KUKA KRL program: MyProgram_329().src

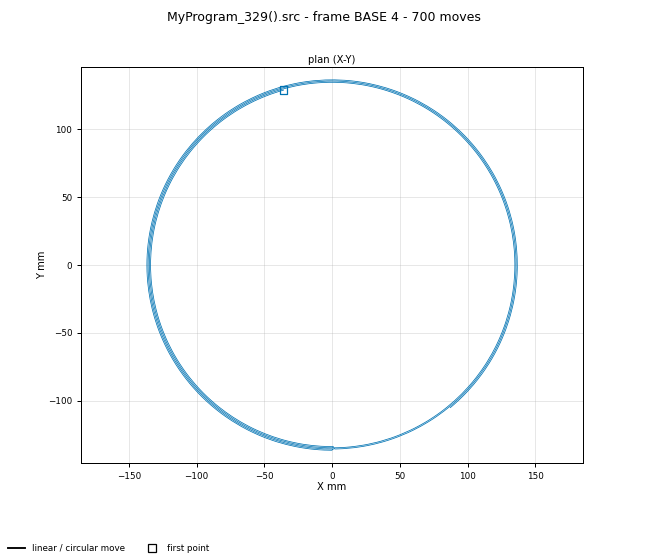
[picture p0: tool path of MyProgram_329().src in frame BASE 4, 700 of 700 moves have a stored position in this frame; points joined in program order, loops and branches not executed]
&ACCESS RVP
&REL 1
&PARAM TEMPLATE = C:\KRC\Roboter\Template\vorgabe
&PARAM EDITMASK = *
DEF MyProgram_329()
; ---- Setting reference (Base) ----
$BASE = BASE_DATA[4]

; --------------------------
; ---- Setting tool (TCP) ----
$TOOL = TOOL_DATA[3]
; --------------------------

$VEL.CP = VEL_APROX_PRINT
Startdeposition()
$VEL.CP = VEL_PRINT
LIN {X -35.8274,Y 129.0295,Z 188,A 105.8967,B 2.405,C -0.0023,E1 2.3658,E2 347.7597} C_DIS
LIN {X -38.989,Y 128.1095,Z 188,A 107.2525,B 2.405,C -0.0012,E1 2.3622,E2 346.4108} C_DIS
LIN {X -42.4339,Y 127.0099,Z 188,A 108.7578,B 2.405,C 0.0001,E1 2.3582,E2 344.9114} C_DIS
LIN {X -45.2331,Y 126.0402,Z 188,A 110.079,B 2.405,C 0.0009,E1 2.3547,E2 343.5846} C_DIS
LIN {X -48.1954,Y 124.9377,Z 188,A 111.532,B 2.405,C 0.0017,E1 2.3509,E2 342.1207} C_DIS
LIN {X -51.2442,Y 123.7186,Z 188,A 112.9196,B 2.405,C 0.003,E1 2.3473,E2 340.736} C_DIS
LIN {X -54.2619,Y 122.4253,Z 188,A 114.3528,B 2.405,C 0.0043,E1 2.3436,E2 339.3003} C_DIS
LIN {X -57.246,Y 121.059,Z 188,A 115.788,B 2.405,C 0.0056,E1 2.3399,E2 337.8624} C_DIS
LIN {X -60.5378,Y 119.4459,Z 188,A 117.3204,B 2.405,C 0.0075,E1 2.3361,E2 336.3352} C_DIS
LIN {X -63.1398,Y 118.0935,Z 188,A 118.6824,B 2.405,C 0.0086,E1 2.3327,E2 334.9616} C_DIS
LIN {X -66.0114,Y 116.513,Z 188,A 120.1274,B 2.405,C 0.0102,E1 2.3292,E2 333.5124} C_DIS
LIN {X -68.8432,Y 114.8624,Z 188,A 121.59,B 2.405,C 0.0118,E1 2.3256,E2 332.0437} C_DIS
LIN {X -71.7353,Y 113.0786,Z 188,A 123.2285,B 2.405,C 0.0132,E1 2.3217,E2 330.3845} C_DIS
LIN {X -74.4991,Y 111.2769,Z 188,A 124.5277,B 2.405,C 0.0156,E1 2.3187,E2 329.0995} C_DIS
LIN {X -77.2049,Y 109.4168,Z 188,A 126.0717,B 2.405,C 0.0172,E1 2.3151,E2 327.5401} C_DIS
LIN {X -80.8265,Y 106.7696,Z 188,A 128.0148,B 2.405,C 0.0201,E1 2.3108,E2 325.5955} C_DIS
LIN {X -83.7272,Y 104.5111,Z 188,A 129.7536,B 2.405,C 0.0222,E1 2.3069,E2 323.8383} C_DIS
LIN {X -86.8424,Y 101.9365,Z 188,A 131.5394,B 2.4049,C 0.025,E1 2.3031,E2 322.0469} C_DIS
LIN {X -89.9692,Y 99.1876,Z 188,A 133.3858,B 2.4049,C 0.028,E1 2.2992,E2 320.194} C_DIS
LIN {X -92.9805,Y 96.3707,Z 188,A 135.2158,B 2.4049,C 0.031,E1 2.2955,E2 318.3575} C_DIS
LIN {X -96.3744,Y 92.9767,Z 188,A 137.2316,B 2.4048,C 0.0351,E1 2.2916,E2 316.3477} C_DIS
LIN {X -99.1765,Y 89.9814,Z 188,A 139.0739,B 2.4048,C 0.0383,E1 2.2881,E2 314.4963} C_DIS
LIN {X -101.9386,Y 86.8399,Z 188,A 140.9329,B 2.4046,C 0.0418,E1 2.2847,E2 312.6304} C_DIS
LIN {X -104.5518,Y 83.676,Z 188,A 142.7551,B 2.4046,C 0.0454,E1 2.2814,E2 310.8016} C_DIS
LIN {X -106.5713,Y 81.0882,Z 188,A 144.2394,B 2.4046,C 0.0482,E1 2.2789,E2 309.3088} C_DIS
LIN {X -108.5268,Y 78.4513,Z 188,A 145.713,B 2.4045,C 0.0511,E1 2.2764,E2 307.828} C_DIS
LIN {X -110.4262,Y 75.7541,Z 188,A 147.2148,B 2.4045,C 0.0541,E1 2.274,E2 306.3165} C_DIS
LIN {X -112.2506,Y 73.0237,Z 188,A 148.7861,B 2.4043,C 0.0569,E1 2.2716,E2 304.7263} C_DIS
LIN {X -114.0716,Y 70.145,Z 188,A 150.2021,B 2.4043,C 0.0604,E1 2.2695,E2 303.3164} C_DIS
LIN {X -115.7605,Y 67.3218,Z 188,A 151.6814,B 2.4042,C 0.0636,E1 2.2674,E2 301.8295} C_DIS
LIN {X -117.3752,Y 64.4659,Z 188,A 153.1513,B 2.4041,C 0.0668,E1 2.2654,E2 300.3527} C_DIS
LIN {X -118.8632,Y 61.6771,Z 188,A 154.6097,B 2.404,C 0.0699,E1 2.2635,E2 298.8825} C_DIS
LIN {X -120.3892,Y 58.6428,Z 188,A 156.2816,B 2.404,C 0.073,E1 2.2614,E2 297.1853} C_DIS
LIN {X -122.2396,Y 54.6771,Z 188,A 158.1986,B 2.4038,C 0.0777,E1 2.2592,E2 295.2642} C_DIS
LIN {X -123.7663,Y 51.1299,Z 188,A 159.8598,B 2.4036,C 0.0819,E1 2.2573,E2 293.6032} C_DIS
LIN {X -125.1601,Y 47.6188,Z 188,A 161.5164,B 2.4035,C 0.086,E1 2.2557,E2 291.9429} C_DIS
LIN {X -126.0828,Y 45.1147,Z 188,A 162.7787,B 2.4034,C 0.0888,E1 2.2544,E2 290.6667} C_DIS
LIN {X -127.1514,Y 42.0088,Z 188,A 164.2678,B 2.4032,C 0.0923,E1 2.2531,E2 289.1686} C_DIS
LIN {X -128.1438,Y 38.8769,Z 188,A 165.7615,B 2.4031,C 0.0959,E1 2.2519,E2 287.6651} C_DIS
LIN {X -129.1832,Y 35.2772,Z 188,A 167.4525,B 2.4029,C 0.1,E1 2.2506,E2 285.9646} C_DIS
LIN {X -129.8894,Y 32.5735,Z 188,A 168.7231,B 2.4029,C 0.1031,E1 2.2497,E2 284.6857} C_DIS
LIN {X -130.6284,Y 29.4706,Z 188,A 170.2306,B 2.4027,C 0.1065,E1 2.2487,E2 283.1616} C_DIS
LIN {X -131.3399,Y 26.122,Z 188,A 171.7271,B 2.4025,C 0.1105,E1 2.2479,E2 281.6622} C_DIS
LIN {X -131.9417,Y 22.8923,Z 188,A 173.3025,B 2.4023,C 0.114,E1 2.2471,E2 280.067} C_DIS
LIN {X -132.4911,Y 19.4568,Z 188,A 174.91,B 2.4021,C 0.1179,E1 2.2464,E2 278.4459} C_DIS
LIN {X -132.9059,Y 16.3864,Z 188,A 176.233,B 2.4019,C 0.1216,E1 2.246,E2 277.124} C_DIS
LIN {X -133.2671,Y 13.1224,Z 188,A 177.7526,B 2.4017,C 0.1253,E1 2.2455,E2 275.5912} C_DIS
LIN {X -133.5485,Y 9.8511,Z 188,A 179.3019,B 2.4016,C 0.1289,E1 2.2452,E2 274.025} C_DIS
LIN {X -133.7561,Y 6.4509,Z 188,A -179.2501,B 2.4013,C 0.1331,E1 2.245,E2 272.5792} C_DIS
LIN {X -133.8718,Y 3.2814,Z 188,A -177.8007,B 2.4011,C 0.1367,E1 2.2448,E2 271.1191} C_DIS
LIN {X -133.9146,Y -0.0043,Z 188,A -176.1985,B 2.4009,C 0.1402,E1 2.2448,E2 269.4936} C_DIS
LIN {X -133.8717,Y -3.2868,Z 188,A -174.7903,B 2.4007,C 0.1442,E1 2.2449,E2 268.0857} C_DIS
LIN {X -133.744,Y -6.6908,Z 188,A -173.2539,B 2.4004,C 0.1481,E1 2.2451,E2 266.5403} C_DIS
LIN {X -133.5487,Y -9.8479,Z 188,A -171.7995,B 2.4002,C 0.1517,E1 2.2454,E2 265.0741} C_DIS
LIN {X -133.2547,Y -13.2522,Z 188,A -170.2718,B 2.4,C 0.1556,E1 2.2458,E2 263.5391} C_DIS
LIN {X -132.8438,Y -16.8815,Z 188,A -168.7185,B 2.3997,C 0.16,E1 2.2463,E2 261.9878} C_DIS
LIN {X -132.446,Y -19.768,Z 188,A -167.259,B 2.3995,C 0.163,E1 2.2469,E2 260.5024} C_DIS
LIN {X -131.9196,Y -23.016,Z 188,A -165.7663,B 2.3992,C 0.1667,E1 2.2476,E2 258.9998} C_DIS
LIN {X -131.314,Y -26.2489,Z 188,A -164.2758,B 2.399,C 0.1704,E1 2.2484,E2 257.4996} C_DIS
LIN {X -130.6304,Y -29.4617,Z 188,A -162.785,B 2.3987,C 0.174,E1 2.2493,E2 255.9987} C_DIS
LIN {X -129.8685,Y -32.6558,Z 188,A -161.1758,B 2.3985,C 0.1774,E1 2.2504,E2 254.3645} C_DIS
LIN {X -128.6799,Y -37.067,Z 188,A -159.1215,B 2.3981,C 0.1824,E1 2.2519,E2 252.2985} C_DIS
LIN {X -127.6271,Y -40.5403,Z 188,A -157.5792,B 2.3978,C 0.1865,E1 2.2532,E2 250.7583} C_DIS
LIN {X -126.3318,Y -44.4155,Z 188,A -155.5541,B 2.3975,C 0.1905,E1 2.2551,E2 248.6988} C_DIS
LIN {X -124.9378,Y -48.1952,Z 188,A -153.9009,B 2.3971,C 0.1951,E1 2.2567,E2 247.0553} C_DIS
LIN {X -123.7177,Y -51.2464,Z 188,A -152.4148,B 2.3968,C 0.1985,E1 2.2583,E2 245.5596} C_DIS
LIN {X -122.4242,Y -54.2643,Z 188,A -150.9184,B 2.3965,C 0.2018,E1 2.2599,E2 244.0521} C_DIS
LIN {X -121.0541,Y -57.2561,Z 188,A -149.4446,B 2.3962,C 0.2052,E1 2.2617,E2 242.5705} C_DIS
LIN {X -119.5578,Y -60.3179,Z 188,A -147.9036,B 2.396,C 0.2086,E1 2.2636,E2 241.0194} C_DIS
LIN {X -118.0969,Y -63.1334,Z 188,A -146.4739,B 2.3957,C 0.2117,E1 2.2655,E2 239.581} C_DIS
LIN {X -116.5142,Y -66.0093,Z 188,A -144.8618,B 2.3954,C 0.2145,E1 2.2677,E2 237.9427} C_DIS
LIN {X -114.2574,Y -69.8422,Z 188,A -142.871,B 2.3951,C 0.2187,E1 2.2706,E2 235.9412} C_DIS
LIN {X -112.2522,Y -73.0211,Z 188,A -141.1446,B 2.3947,C 0.2221,E1 2.2732,E2 234.2} C_DIS
LIN {X -109.6344,Y -76.8963,Z 188,A -139.1029,B 2.3943,C 0.2264,E1 2.2765,E2 232.1536} C_DIS
LIN {X -107.4833,Y -79.8748,Z 188,A -137.4158,B 2.394,C 0.2295,E1 2.2793,E2 230.4519} C_DIS
LIN {X -105.0604,Y -83.0368,Z 188,A -135.7516,B 2.3937,C 0.2332,E1 2.2821,E2 228.7934} C_DIS
LIN {X -102.9533,Y -85.6349,Z 188,A -134.1037,B 2.3935,C 0.2355,E1 2.2851,E2 227.1177} C_DIS
LIN {X -100.8628,Y -88.0871,Z 188,A -132.8082,B 2.3932,C 0.2386,E1 2.2875,E2 225.8332} C_DIS
LIN {X -98.1094,Y -91.1439,Z 188,A -130.9727,B 2.3928,C 0.2418,E1 2.291,E2 223.9882} C_DIS
LIN {X -95.2718,Y -94.1067,Z 188,A -129.1535,B 2.3925,C 0.2449,E1 2.2945,E2 222.1609} C_DIS
LIN {X -92.3885,Y -96.9383,Z 188,A -127.3391,B 2.3922,C 0.2478,E1 2.2982,E2 220.3357} C_DIS
LIN {X -89.3651,Y -99.7322,Z 188,A -125.4998,B 2.3919,C 0.2507,E1 2.302,E2 218.4863} C_DIS
LIN {X -86.2189,Y -102.4645,Z 188,A -123.6636,B 2.3916,C 0.2535,E1 2.3059,E2 216.6433} C_DIS
LIN {X -83.6332,Y -104.5859,Z 188,A -122.0545,B 2.3914,C 0.2552,E1 2.3095,E2 215.011} C_DIS
LIN {X -80.6086,Y -106.9341,Z 188,A -120.617,B 2.3911,C 0.2585,E1 2.3126,E2 213.5997} C_DIS
LIN {X -78.4436,Y -108.5323,Z 188,A -119.2375,B 2.391,C 0.2594,E1 2.3158,E2 212.1904} C_DIS
LIN {X -75.7529,Y -110.427,Z 188,A -117.8311,B 2.3908,C 0.2614,E1 2.319,E2 210.7842} C_DIS
LIN {X -73.025,Y -112.2497,Z 188,A -116.4108,B 2.3906,C 0.2633,E1 2.3223,E2 209.3617} C_DIS
LIN {X -70.1501,Y -114.0685,Z 188,A -114.8476,B 2.3904,C 0.2648,E1 2.3261,E2 207.7843} C_DIS
LIN {X -67.3364,Y -115.752,Z 188,A -113.4736,B 2.3902,C 0.2667,E1 2.3294,E2 206.414} C_DIS
LIN {X -64.4813,Y -117.3668,Z 188,A -111.8722,B 2.3901,C 0.2676,E1 2.3334,E2 204.7864} C_DIS
LIN {X -61.6733,Y -118.8651,Z 188,A -110.6199,B 2.3899,C 0.2696,E1 2.3364,E2 203.5483} C_DIS
LIN {X -58.62,Y -120.4004,Z 188,A -109.1295,B 2.3897,C 0.271,E1 2.3402,E2 202.054} C_DIS
LIN {X -55.6518,Y -121.8004,Z 188,A -107.6966,B 2.3896,C 0.2723,E1 2.3438,E2 200.6171} C_DIS
LIN {X -52.591,Y -123.1529,Z 188,A -106.2406,B 2.3894,C 0.2735,E1 2.3476,E2 199.1576} C_DIS
LIN {X -49.6154,Y -124.3811,Z 188,A -104.775,B 2.3894,C 0.2743,E1 2.3514,E2 197.6801} C_DIS
LIN {X -46.1766,Y -125.7,Z 188,A -103.2397,B 2.3892,C 0.2758,E1 2.3554,E2 196.1498} C_DIS
LIN {X -43.5843,Y -126.62,Z 188,A -102.0049,B 2.3891,C 0.2764,E1 2.3587,E2 194.9071} C_DIS
LIN {X -40.439,Y -127.6594,Z 188,A -100.6013,B 2.389,C 0.2774,E1 2.3624,E2 193.5049} C_DIS
LIN {X -37.2954,Y -128.613,Z 188,A -99.1783,B 2.3889,C 0.2782,E1 2.3663,E2 192.0793} C_DIS
LIN {X -34.1281,Y -129.4897,Z 188,A -97.7576,B 2.3889,C 0.2788,E1 2.3701,E2 190.6562} C_DIS
LIN {X -30.2809,Y -130.4433,Z 188,A -96.1746,B 2.3886,C 0.2802,E1 2.3744,E2 189.0875} C_DIS
LIN {X -27.0839,Y -131.1441,Z 188,A -94.7939,B 2.3886,C 0.2808,E1 2.3781,E2 187.709} C_DIS
LIN {X -24.514,Y -131.6497,Z 188,A -93.4398,B 2.3886,C 0.28,E1 2.382,E2 186.3237} C_DIS
LIN {X -21.2716,Y -132.2131,Z 188,A -92.0361,B 2.3886,C 0.2804,E1 2.3858,E2 184.9201} C_DIS
LIN {X -17.749,Y -132.7302,Z 188,A -90.6329,B 2.3886,C 0.2813,E1 2.3897,E2 183.5321} C_DIS
LIN {X -14.7665,Y -133.0953,Z 188,A -89.2585,B 2.3886,C 0.281,E1 2.3935,E2 182.1454} C_DIS
LIN {X -11.3769,Y -133.4271,Z 188,A -87.832,B 2.3886,C 0.2812,E1 2.3975,E2 180.7225} C_DIS
LIN {X -8.2084,Y -133.6595,Z 188,A -86.4352,B 2.3886,C 0.281,E1 2.4014,E2 179.3201} C_DIS
LIN {X -4.8094,Y -133.8255,Z 188,A -85.0219,B 2.3886,C 0.2811,E1 2.4053,E2 177.9118} C_DIS
LIN {X -1.5336,Y -133.9044,Z 188,A -83.6281,B 2.3886,C 0.2809,E1 2.4092,E2 176.5184} C_DIS
LIN {X 0.9694,Y -133.9063,Z 188,A -82.8484,B 2.3884,C 0.2824,E1 2.4113,E2 175.7765} C_DIS
Enddeposition()
LIN {X 0.9694,Y -133.9063,Z 188,A -82.8484,B 2.3884,C 0.2824,E1 2.4113,E2 175.7765} C_DIS
Startdeposition()
$VEL.CP = VEL_PRINT
LIN {X 0.415,Y -134.8105,Z 188,A -83.4457,B 2.388,C 0.2858,E1 2.4095,E2 176.4517} C_DIS
LIN {X -3.4942,Y -134.7656,Z 188,A -85.0636,B 2.388,C 0.2858,E1 2.405,E2 178.0646} C_DIS
LIN {X -7.3404,Y -134.6118,Z 188,A -86.8771,B 2.388,C 0.2869,E1 2.3998,E2 179.9022} C_DIS
LIN {X -12.0577,Y -134.2721,Z 188,A -88.6303,B 2.388,C 0.2854,E1 2.395,E2 181.6224} C_DIS
LIN {X -15.2807,Y -133.9435,Z 188,A -89.9903,B 2.388,C 0.2852,E1 2.3913,E2 182.9808} C_DIS
LIN {X -19.8517,Y -133.3431,Z 188,A -92.1758,B 2.388,C 0.286,E1 2.3851,E2 185.1969} C_DIS
LIN {X -24.3404,Y -132.5962,Z 188,A -94.0832,B 2.388,C 0.2854,E1 2.3799,E2 187.1015} C_DIS
LIN {X -28.5188,Y -131.7593,Z 188,A -95.7935,B 2.3882,C 0.2842,E1 2.3752,E2 188.799} C_DIS
LIN {X -31.6082,Y -131.0525,Z 188,A -97.2414,B 2.3882,C 0.2841,E1 2.3712,E2 190.2606} C_DIS
LIN {X -35.3493,Y -130.0948,Z 188,A -98.8051,B 2.3884,C 0.2828,E1 2.367,E2 191.8147} C_DIS
LIN {X -38.0908,Y -129.3172,Z 188,A -100.0429,B 2.3884,C 0.2823,E1 2.3637,E2 193.0563} C_DIS
LIN {X -41.0419,Y -128.4109,Z 188,A -101.4355,B 2.3885,C 0.2818,E1 2.3599,E2 194.4599} C_DIS
LIN {X -47.3357,Y -126.2264,Z 188,A -103.8946,B 2.3889,C 0.278,E1 2.3536,E2 196.8706} C_DIS
LIN {X -49.902,Y -125.2352,Z 188,A -105.3116,B 2.3889,C 0.2781,E1 2.3498,E2 198.3206} C_DIS
LIN {X -52.2633,Y -124.2676,Z 188,A -106.6515,B 2.3889,C 0.2783,E1 2.3462,E2 199.6943} C_DIS
LIN {X -55.7004,Y -122.767,Z 188,A -108.3329,B 2.389,C 0.2771,E1 2.3419,E2 201.3874} C_DIS
LIN {X -59.6229,Y -120.9085,Z 188,A -110.0185,B 2.3893,C 0.2745,E1 2.3377,E2 203.0525} C_DIS
LIN {X -63.0785,Y -119.143,Z 188,A -111.7381,B 2.3895,C 0.273,E1 2.3334,E2 204.7815} C_DIS
LIN {X -67.1827,Y -116.8801,Z 188,A -113.8146,B 2.3898,C 0.2709,E1 2.3283,E2 206.8694} C_DIS
LIN {X -70.5116,Y -114.9018,Z 188,A -115.5702,B 2.39,C 0.2692,E1 2.3241,E2 208.6394} C_DIS
LIN {X -74.1577,Y -112.583,Z 188,A -117.4112,B 2.3902,C 0.2667,E1 2.3198,E2 210.4811} C_DIS
LIN {X -77.6689,Y -110.19,Z 188,A -119.1037,B 2.3906,C 0.2637,E1 2.3159,E2 212.1588} C_DIS
LIN {X -80.1343,Y -108.411,Z 188,A -120.6784,B 2.3906,C 0.2628,E1 2.3123,E2 213.7704} C_DIS
LIN {X -83.6524,Y -105.7201,Z 188,A -122.6514,B 2.391,C 0.2602,E1 2.3079,E2 215.7552} C_DIS
LIN {X -87.0884,Y -102.9077,Z 188,A -124.5819,B 2.3913,C 0.2572,E1 2.3037,E2 217.6912} C_DIS
LIN {X -90.4103,Y -100.0017,Z 188,A -126.5158,B 2.3916,C 0.2541,E1 2.2997,E2 219.6325} C_DIS
LIN {X -93.6298,Y -96.9938,Z 188,A -128.3841,B 2.392,C 0.2507,E1 2.2959,E2 221.5} C_DIS
LIN {X -96.1827,Y -94.4626,Z 188,A -129.9743,B 2.3922,C 0.248,E1 2.2927,E2 223.0982} C_DIS
LIN {X -98.6686,Y -91.863,Z 188,A -131.7171,B 2.3925,C 0.2458,E1 2.2893,E2 224.8684} C_DIS
LIN {X -101.8246,Y -88.3526,Z 188,A -133.5778,B 2.3929,C 0.2413,E1 2.2859,E2 226.71} C_DIS
LIN {X -104.0657,Y -85.7015,Z 188,A -135.2736,B 2.3932,C 0.2389,E1 2.2828,E2 228.4339} C_DIS
LIN {X -106.7775,Y -82.2982,Z 188,A -137.2732,B 2.3935,C 0.2355,E1 2.2793,E2 230.4525} C_DIS
LIN {X -109.1126,Y -79.1755,Z 188,A -138.9644,B 2.3939,C 0.232,E1 2.2765,E2 232.1476} C_DIS
LIN {X -111.7399,Y -75.4224,Z 188,A -141.0239,B 2.3942,C 0.2279,E1 2.2733,E2 234.221} C_DIS
LIN {X -114.2514,Y -71.5617,Z 188,A -142.9088,B 2.3947,C 0.2232,E1 2.2704,E2 236.0961} C_DIS
LIN {X -116.0683,Y -68.5753,Z 188,A -144.5383,B 2.395,C 0.2202,E1 2.2681,E2 237.7437} C_DIS
LIN {X -117.5639,Y -65.9776,Z 188,A -145.7805,B 2.3953,C 0.217,E1 2.2663,E2 238.9814} C_DIS
LIN {X -118.7226,Y -63.869,Z 188,A -147.0145,B 2.3954,C 0.2151,E1 2.2647,E2 240.242} C_DIS
LIN {X -120.2859,Y -60.87,Z 188,A -148.4629,B 2.3957,C 0.2116,E1 2.2628,E2 241.6912} C_DIS
LIN {X -121.6873,Y -58.0169,Z 188,A -149.8404,B 2.396,C 0.2084,E1 2.2611,E2 243.0716} C_DIS
LIN {X -123.1403,Y -54.866,Z 188,A -151.484,B 2.3963,C 0.2051,E1 2.2592,E2 244.7362} C_DIS
LIN {X -124.4666,Y -51.7867,Z 188,A -152.9088,B 2.3966,C 0.2015,E1 2.2577,E2 246.1604} C_DIS
LIN {X -125.6422,Y -48.8652,Z 188,A -154.3937,B 2.3969,C 0.1984,E1 2.2561,E2 247.6632} C_DIS
LIN {X -127.003,Y -45.2143,Z 188,A -156.0756,B 2.3972,C 0.1941,E1 2.2545,E2 249.3478} C_DIS
LIN {X -129.2375,Y -38.3631,Z 188,A -159.2378,B 2.3978,C 0.1863,E1 2.2518,E2 252.5212} C_DIS
LIN {X -130.3562,Y -34.3687,Z 188,A -161.235,B 2.3982,C 0.182,E1 2.2503,E2 254.5472} C_DIS
LIN {X -131.1326,Y -31.2758,Z 188,A -162.6422,B 2.3984,C 0.1785,E1 2.2493,E2 255.9603} C_DIS
LIN {X -131.7871,Y -28.3903,Z 188,A -164.0512,B 2.3987,C 0.1754,E1 2.2485,E2 257.3876} C_DIS
LIN {X -132.618,Y -24.2188,Z 188,A -166.0152,B 2.399,C 0.1708,E1 2.2474,E2 259.3702} C_DIS
LIN {X -133.2441,Y -20.4914,Z 188,A -167.6839,B 2.3993,C 0.1664,E1 2.2467,E2 261.0458} C_DIS
LIN {X -133.7144,Y -17.1595,Z 188,A -169.1662,B 2.3996,C 0.1626,E1 2.2461,E2 262.5338} C_DIS
LIN {X -134.0775,Y -14.0441,Z 188,A -170.7279,B 2.3998,C 0.1594,E1 2.2457,E2 264.1233} C_DIS
LIN {X -134.4509,Y -9.8412,Z 188,A -172.5175,B 2.4001,C 0.1543,E1 2.2453,E2 265.9113} C_DIS
LIN {X -134.6645,Y -6.2931,Z 188,A -174.0277,B 2.4004,C 0.1501,E1 2.245,E2 267.4206} C_DIS
LIN {X -134.768,Y -3.4066,Z 188,A -175.4035,B 2.4006,C 0.147,E1 2.245,E2 268.8141} C_DIS
LIN {X -134.8108,Y 0.5522,Z 188,A -177.3255,B 2.4008,C 0.1427,E1 2.2449,E2 270.7646} C_DIS
LIN {X -134.7107,Y 5.191,Z 188,A -179.3112,B 2.4011,C 0.1372,E1 2.245,E2 272.7507} C_DIS
LIN {X -134.5409,Y 8.5264,Z 188,A 179.0777,B 2.4013,C 0.1336,E1 2.2453,E2 274.3845} C_DIS
LIN {X -134.2141,Y 12.6695,Z 188,A 177.1896,B 2.4016,C 0.1289,E1 2.2458,E2 276.2864} C_DIS
LIN {X -133.722,Y 17.1021,Z 188,A 175.1938,B 2.4019,C 0.1238,E1 2.2464,E2 278.2933} C_DIS
LIN {X -133.1367,Y 21.1846,Z 188,A 173.4587,B 2.4021,C 0.1189,E1 2.2471,E2 280.025} C_DIS
LIN {X -132.6136,Y 24.2431,Z 188,A 172.0685,B 2.4023,C 0.1154,E1 2.2478,E2 281.423} C_DIS
LIN {X -131.8998,Y 27.8682,Z 188,A 169.5957,B 2.4024,C 0.113,E1 2.2493,E2 284.0042} C_DIS
LIN {X -130.6708,Y 33.1506,Z 188,A 167.864,B 2.4027,C 0.1055,E1 2.2504,E2 285.665} C_DIS
LIN {X -129.6037,Y 37.1124,Z 188,A 165.8558,B 2.4029,C 0.1014,E1 2.252,E2 287.7041} C_DIS
LIN {X -128.3694,Y 41.1719,Z 188,A 164.0931,B 2.4031,C 0.0964,E1 2.2534,E2 289.4605} C_DIS
LIN {X -127.3513,Y 44.2205,Z 188,A 162.703,B 2.4033,C 0.0929,E1 2.2547,E2 290.8525} C_DIS
LIN {X -126.0119,Y 47.9086,Z 188,A 160.953,B 2.4034,C 0.0887,E1 2.2564,E2 292.6113} C_DIS
LIN {X -124.6936,Y 51.2433,Z 188,A 159.1647,B 2.4035,C 0.0853,E1 2.2583,E2 294.4304} C_DIS
LIN {X -122.4485,Y 56.393,Z 188,A 157.0175,B 2.4038,C 0.0787,E1 2.2607,E2 296.5468} C_DIS
LIN {X -121.4634,Y 58.4857,Z 188,A 155.7507,B 2.4038,C 0.0769,E1 2.2622,E2 297.8471} C_DIS
LIN {X -119.6333,Y 62.1447,Z 188,A 154.0252,B 2.404,C 0.0726,E1 2.2644,E2 299.5698} C_DIS
LIN {X -117.4103,Y 66.2508,Z 188,A 151.8315,B 2.404,C 0.0682,E1 2.2674,E2 301.7871} C_DIS
LIN {X -115.489,Y 69.5462,Z 188,A 150.0107,B 2.4042,C 0.0648,E1 2.27,E2 303.6306} C_DIS
LIN {X -113.299,Y 73.0603,Z 188,A 148.2346,B 2.4042,C 0.0608,E1 2.2727,E2 305.4073} C_DIS
LIN {X -110.9551,Y 76.5728,Z 188,A 146.3565,B 2.4044,C 0.0569,E1 2.2756,E2 307.294} C_DIS
LIN {X -108.5031,Y 80.009,Z 188,A 144.5849,B 2.4044,C 0.0529,E1 2.2785,E2 309.0616} C_DIS
LIN {X -106.9738,Y 82.0422,Z 188,A 143.455,B 2.4045,C 0.0506,E1 2.2804,E2 310.1964} C_DIS
LIN {X -104.9898,Y 84.5662,Z 188,A 141.8919,B 2.4045,C 0.0482,E1 2.2832,E2 311.7821} C_DIS
LIN {X -102.2723,Y 87.8334,Z 188,A 139.9216,B 2.4046,C 0.0449,E1 2.2868,E2 313.7705} C_DIS
LIN {X -98.8639,Y 91.6533,Z 188,A 137.6428,B 2.4047,C 0.0408,E1 2.2911,E2 316.0599} C_DIS
LIN {X -95.6921,Y 94.9596,Z 188,A 135.633,B 2.4047,C 0.0372,E1 2.295,E2 318.0756} C_DIS
LIN {X -92.2591,Y 98.2989,Z 188,A 133.5112,B 2.4048,C 0.0337,E1 2.2993,E2 320.2061} C_DIS
LIN {X -88.9181,Y 101.3312,Z 188,A 131.5845,B 2.4048,C 0.0303,E1 2.3033,E2 322.1325} C_DIS
LIN {X -86.1319,Y 103.7094,Z 188,A 129.9774,B 2.4048,C 0.0278,E1 2.3068,E2 323.7444} C_DIS
LIN {X -83.2724,Y 106.0189,Z 188,A 128.38,B 2.4049,C 0.0254,E1 2.3103,E2 325.3448} C_DIS
LIN {X -79.474,Y 108.8961,Z 188,A 126.3051,B 2.4049,C 0.0223,E1 2.3149,E2 327.4242} C_DIS
LIN {X -76.336,Y 111.1176,Z 188,A 124.6083,B 2.4049,C 0.0201,E1 2.3188,E2 329.1272} C_DIS
LIN {X -73.7185,Y 112.8717,Z 188,A 122.9421,B 2.4049,C 0.0193,E1 2.3228,E2 330.8307} C_DIS
LIN {X -69.3256,Y 115.6218,Z 188,A 120.8519,B 2.405,C 0.0159,E1 2.3278,E2 332.9063} C_DIS
LIN {X -66.003,Y 117.5496,Z 188,A 119.0641,B 2.405,C 0.0144,E1 2.3322,E2 334.7111} C_DIS
LIN {X -61.2031,Y 120.1163,Z 188,A 116.8852,B 2.405,C 0.0112,E1 2.3375,E2 336.8728} C_DIS
LIN {X -57.531,Y 121.9195,Z 188,A 115.1134,B 2.405,C 0.0094,E1 2.342,E2 338.6475} C_DIS
LIN {X -54.4451,Y 123.3285,Z 188,A 113.6869,B 2.405,C 0.0079,E1 2.3456,E2 340.0712} C_DIS
LIN {X -51.179,Y 124.7204,Z 188,A 112.116,B 2.405,C 0.0068,E1 2.3497,E2 341.6485} C_DIS
LIN {X -47.8265,Y 126.0426,Z 188,A 110.6562,B 2.405,C 0.0051,E1 2.3535,E2 343.0989} C_DIS
LIN {X -44.8357,Y 127.138,Z 188,A 108.9366,B 2.405,C 0.0055,E1 2.3581,E2 344.8603} C_DIS
LIN {X -40.0632,Y 128.7212,Z 188,A 106.8723,B 2.405,C 0.0037,E1 2.3636,E2 346.9149} C_DIS
LIN {X -36.2129,Y 129.8555,Z 188,A 105.2751,B 2.405,C 0.0022,E1 2.3678,E2 348.4984} C_DIS
LIN {X -32.9402,Y 130.7242,Z 188,A 103.8802,B 2.405,C 0.0012,E1 2.3716,E2 349.8875} C_DIS
LIN {X -29.3217,Y 131.5849,Z 188,A 102.2423,B 2.405,C 0.0007,E1 2.3761,E2 351.5312} C_DIS
LIN {X -26.6535,Y 132.1495,Z 188,A 101.0267,B 2.405,C 0.0005,E1 2.3794,E2 352.7527} C_DIS
LIN {X -22.4807,Y 132.9231,Z 188,A 99.0934,B 2.405,C 0.0005,E1 2.3848,E2 354.7} C_DIS
LIN {X -17.5729,Y 133.6603,Z 188,A 97.0368,B 2.405,C -0.0002,E1 2.3905,E2 356.7495} C_DIS
LIN {X -13.9523,Y 134.0874,Z 188,A 95.4131,B 2.405,C -0.0001,E1 2.395,E2 358.3811} C_DIS
LIN {X -10.2269,Y 134.4227,Z 188,A 93.892,B 2.405,C -0.0005,E1 2.3992,E2 359.8935} C_DIS
LIN {X -5.4082,Y 134.7022,Z 188,A 92.1825,B 2.405,C -0.0021,E1 2.4039,E2 361.5624} C_DIS
LIN {X -2.4079,Y 134.7893,Z 188,A 90.5819,B 2.405,C -0.0004,E1 2.4085,E2 363.2003} C_DIS
LIN {X 2.0008,Y 134.796,Z 188,A 88.7247,B 2.405,C -0.0001,E1 2.4137,E2 365.0548} C_DIS
LIN {X 6.3924,Y 134.6595,Z 188,A 86.7805,B 2.405,C 0.0008,E1 2.4191,E2 367.0071} C_DIS
LIN {X 10.5609,Y 134.3983,Z 188,A 84.9962,B 2.405,C 0.0015,E1 2.4241,E2 368.7919} C_DIS
LIN {X 14.9972,Y 133.975,Z 188,A 83.2838,B 2.405,C 0.0014,E1 2.4288,E2 370.4825} C_DIS
LIN {X 19.1062,Y 133.4497,Z 188,A 81.6138,B 2.405,C 0.0018,E1 2.4334,E2 372.1414} C_DIS
LIN {X 21.9585,Y 133.0103,Z 188,A 80.2361,B 2.405,C 0.0034,E1 2.4373,E2 373.5363} C_DIS
LIN {X 25.6226,Y 132.3534,Z 188,A 78.7143,B 2.405,C 0.0041,E1 2.4414,E2 375.0505} C_DIS
LIN {X 29.997,Y 131.4306,Z 188,A 76.8943,B 2.405,C 0.0051,E1 2.4464,E2 376.8607} C_DIS
LIN {X 33.6535,Y 130.5432,Z 188,A 75.3617,B 2.405,C 0.0061,E1 2.4505,E2 378.3851} C_DIS
LIN {X 36.7136,Y 129.7154,Z 188,A 74.0913,B 2.405,C 0.0068,E1 2.4539,E2 379.6463} C_DIS
LIN {X 40.0229,Y 128.7335,Z 188,A 72.0606,B 2.405,C 0.0116,E1 2.4595,E2 381.7422} C_DIS
LIN {X 44.1717,Y 127.3682,Z 188,A 71.0763,B 2.405,C 0.0083,E1 2.4619,E2 382.6245} C_DIS
LIN {X 47.0616,Y 126.3291,Z 188,A 69.6449,B 2.405,C 0.0105,E1 2.4657,E2 384.0704} C_DIS
LIN {X 49.2176,Y 125.5052,Z 188,A 68.3938,B 2.405,C 0.0133,E1 2.469,E2 385.3531} C_DIS
LIN {X 52.6088,Y 124.1233,Z 188,A 66.8377,B 2.405,C 0.0152,E1 2.473,E2 386.9089} C_DIS
LIN {X 56.8704,Y 122.2277,Z 188,A 64.9766,B 2.405,C 0.017,E1 2.4777,E2 388.7556} C_DIS
LIN {X 60.2635,Y 120.5925,Z 188,A 63.5212,B 2.405,C 0.0183,E1 2.4814,E2 390.1938} C_DIS
LIN {X 65.4535,Y 117.8566,Z 188,A 61.2376,B 2.405,C 0.0205,E1 2.4869,E2 392.4525} C_DIS
LIN {X 68.2924,Y 116.2345,Z 188,A 59.6873,B 2.405,C 0.0237,E1 2.4907,E2 394.0216} C_DIS
LIN {X 71.9286,Y 114.0201,Z 188,A 57.9398,B 2.405,C 0.0262,E1 2.4949,E2 395.7617} C_DIS
LIN {X 74.6265,Y 112.2731,Z 188,A 56.6318,B 2.4049,C 0.028,E1 2.4979,E2 397.0628} C_DIS
LIN {X 78.0883,Y 109.8939,Z 188,A 54.8511,B 2.4049,C 0.0311,E1 2.502,E2 398.843} C_DIS
LIN {X 81.7113,Y 107.227,Z 188,A 53.0922,B 2.4049,C 0.0334,E1 2.5059,E2 400.5839} C_DIS
LIN {X 84.8107,Y 104.7927,Z 188,A 51.4568,B 2.4048,C 0.0362,E1 2.5094,E2 402.2146} C_DIS
LIN {X 87.9293,Y 102.1897,Z 188,A 49.7869,B 2.4048,C 0.0391,E1 2.513,E2 403.8779} C_DIS
LIN {X 92.3112,Y 98.2498,Z 188,A 47.3591,B 2.4047,C 0.0436,E1 2.518,E2 406.2969} C_DIS
LIN {X 95.4989,Y 95.154,Z 188,A 45.4471,B 2.4046,C 0.0476,E1 2.5218,E2 408.2119} C_DIS
LIN {X 98.8526,Y 91.6654,Z 188,A 43.61,B 2.4046,C 0.0503,E1 2.5253,E2 410.0231} C_DIS
LIN {X 101.6038,Y 88.6057,Z 188,A 41.9522,B 2.4045,C 0.0535,E1 2.5283,E2 411.6703} C_DIS
LIN {X 104.2348,Y 85.4954,Z 188,A 40.2803,B 2.4044,C 0.0569,E1 2.5313,E2 413.3355} C_DIS
LIN {X 106.8063,Y 82.2611,Z 188,A 38.5611,B 2.4043,C 0.0606,E1 2.5343,E2 415.0506} C_DIS
LIN {X 109.0567,Y 79.2526,Z 188,A 37.0496,B 2.4043,C 0.0636,E1 2.5367,E2 416.5522} C_DIS
LIN {X 112.1603,Y 74.7955,Z 188,A 34.8989,B 2.4041,C 0.0679,E1 2.5401,E2 418.6845} C_DIS
LIN {X 114.5673,Y 71.0541,Z 188,A 33.1244,B 2.404,C 0.0716,E1 2.5428,E2 420.4455} C_DIS
LIN {X 116.968,Y 67.0289,Z 188,A 31.1881,B 2.4039,C 0.076,E1 2.5455,E2 422.3758} C_DIS
LIN {X 118.6791,Y 63.95,Z 188,A 29.7687,B 2.4038,C 0.0792,E1 2.5474,E2 423.7862} C_DIS
LIN {X 120.3947,Y 60.6563,Z 188,A 28.2411,B 2.4036,C 0.0828,E1 2.5493,E2 425.3082} C_DIS
LIN {X 121.9341,Y 57.5004,Z 188,A 26.943,B 2.4036,C 0.085,E1 2.5508,E2 426.5832} C_DIS
LIN {X 123.46,Y 54.1469,Z 188,A 25.485,B 2.4034,C 0.0882,E1 2.5525,E2 428.0287} C_DIS
LIN {X 124.9152,Y 50.6959,Z 188,A 23.4646,B 2.4031,C 0.0958,E1 2.5547,E2 430.1018} C_DIS
LIN {X 126.4955,Y 46.6174,Z 188,A 21.9697,B 2.4031,C 0.0978,E1 2.5561,E2 431.5532} C_DIS
LIN {X 127.8806,Y 42.6656,Z 188,A 20.4415,B 2.403,C 0.1006,E1 2.5575,E2 433.0514} C_DIS
LIN {X 129.0066,Y 39.1307,Z 188,A 18.9724,B 2.4028,C 0.1039,E1 2.5587,E2 434.5081} C_DIS
LIN {X 129.9056,Y 36.0335,Z 188,A 17.7317,B 2.4027,C 0.1066,E1 2.5596,E2 435.7334} C_DIS
LIN {X 130.7401,Y 32.8776,Z 188,A 16.4194,B 2.4026,C 0.1098,E1 2.5605,E2 437.0372} C_DIS
LIN {X 131.4867,Y 29.7517,Z 188,A 15.1052,B 2.4024,C 0.1131,E1 2.5614,E2 438.3457} C_DIS
LIN {X 132.209,Y 26.3608,Z 188,A 13.7302,B 2.4022,C 0.1164,E1 2.5621,E2 439.7093} C_DIS
LIN {X 132.7592,Y 23.4299,Z 188,A 12.405,B 2.402,C 0.1203,E1 2.5628,E2 441.0423} C_DIS
LIN {X 133.365,Y 19.6987,Z 188,A 11.057,B 2.402,C 0.1227,E1 2.5634,E2 442.3591} C_DIS
LIN {X 133.7685,Y 16.7467,Z 188,A 9.5885,B 2.4017,C 0.1279,E1 2.5639,E2 443.8535} C_DIS
LIN {X 134.308,Y 11.6336,Z 188,A 7.9204,B 2.4016,C 0.1297,E1 2.5643,E2 445.4585} C_DIS
LIN {X 134.5504,Y 8.3729,Z 188,A 6.351,B 2.4013,C 0.1351,E1 2.5646,E2 447.0512} C_DIS
LIN {X 134.7191,Y 4.9741,Z 188,A 5.0443,B 2.4011,C 0.138,E1 2.5648,E2 448.3413} C_DIS
LIN {X 134.8105,Y 0.6078,Z 188,A 3.2534,B 2.4008,C 0.1427,E1 2.5648,E2 450.1253} C_DIS
LIN {X 134.7632,Y -3.5807,Z 188,A 1.5234,B 2.4005,C 0.1472,E1 2.5648,E2 451.8501} C_DIS
LIN {X 134.62,Y -7.179,Z 188,A 0.2169,B 2.4004,C 0.1497,E1 2.5646,E2 453.1295} C_DIS
LIN {X 134.3764,Y -10.8231,Z 188,A -1.1852,B 2.4002,C 0.1528,E1 2.5643,E2 454.5137} C_DIS
LIN {X 134.0875,Y -13.9512,Z 188,A -2.4364,B 2.4,C 0.1558,E1 2.564,E2 455.7553} C_DIS
LIN {X 133.8005,Y -16.4788,Z 188,A -3.5137,B 2.3998,C 0.1588,E1 2.5637,E2 456.8328} C_DIS
LIN {X 133.4429,Y -19.1536,Z 188,A -4.5827,B 2.3996,C 0.1613,E1 2.5633,E2 457.8927} C_DIS
LIN {X 132.925,Y -22.4692,Z 188,A -6.032,B 2.3994,C 0.1655,E1 2.5626,E2 459.3459} C_DIS
LIN {X 132.0588,Y -27.0991,Z 188,A -7.8956,B 2.3991,C 0.1699,E1 2.5616,E2 461.1934} C_DIS
LIN {X 131.2812,Y -30.651,Z 188,A -9.4804,B 2.3987,C 0.1745,E1 2.5606,E2 462.7843} C_DIS
LIN {X 130.1693,Y -35.0697,Z 188,A -11.2558,B 2.3984,C 0.1784,E1 2.5594,E2 464.5407} C_DIS
LIN {X 128.1562,Y -41.838,Z 188,A -14.0149,B 2.398,C 0.1846,E1 2.5572,E2 467.2713} C_DIS
LIN {X 127.1714,Y -44.7393,Z 188,A -15.2681,B 2.3977,C 0.1876,E1 2.5561,E2 468.5192} C_DIS
LIN {X 125.5609,Y -49.0745,Z 188,A -17.1446,B 2.3974,C 0.1921,E1 2.5542,E2 470.3858} C_DIS
LIN {X 123.6513,Y -53.7046,Z 188,A -19.1981,B 2.397,C 0.1971,E1 2.552,E2 472.4313} C_DIS
LIN {X 122.1914,Y -56.949,Z 188,A -20.5523,B 2.3968,C 0.1997,E1 2.5504,E2 473.7664} C_DIS
LIN {X 120.7468,Y -59.9508,Z 188,A -21.9739,B 2.3964,C 0.2034,E1 2.5487,E2 475.1898} C_DIS
LIN {X 118.0966,Y -65.0201,Z 188,A -24.3496,B 2.396,C 0.2091,E1 2.5456,E2 477.5604} C_DIS
LIN {X 115.7695,Y -69.0778,Z 188,A -26.0097,B 2.3958,C 0.2113,E1 2.5433,E2 479.1799} C_DIS
LIN {X 114.5027,Y -71.1578,Z 188,A -27.0197,B 2.3956,C 0.2137,E1 2.5418,E2 480.1875} C_DIS
LIN {X 113.131,Y -73.3192,Z 188,A -28.1949,B 2.3953,C 0.217,E1 2.54,E2 481.3748} C_DIS
LIN {X 110.5006,Y -77.2268,Z 188,A -30.9898,B 2.3942,C 0.2281,E1 2.5354,E2 484.2728} C_DIS
LIN {X 106.3482,Y -82.8521,Z 188,A -32.9403,B 2.3943,C 0.2269,E1 2.5323,E2 486.0947} C_DIS
LIN {X 103.5929,Y -86.2725,Z 188,A -35.1584,B 2.3937,C 0.2338,E1 2.5283,E2 488.3596} C_DIS
LIN {X 100.6702,Y -89.6657,Z 188,A -36.3088,B 2.3938,C 0.2321,E1 2.5264,E2 489.4141} C_DIS
LIN {X 95.8069,Y -94.8441,Z 188,A -39.446,B 2.3931,C 0.2395,E1 2.5203,E2 492.5691} C_DIS
LIN {X 90.5199,Y -99.9022,Z 188,A -42.2126,B 2.3927,C 0.2432,E1 2.5148,E2 495.2936} C_DIS
LIN {X 84.7789,Y -104.8183,Z 188,A -46.0124,B 2.3916,C 0.2538,E1 2.5064,E2 499.1723} C_DIS
LIN {X 80.9116,Y -107.832,Z 188,A -47.4163,B 2.3918,C 0.2525,E1 2.5035,E2 500.4894} C_DIS
LIN {X 78.144,Y -109.8541,Z 188,A -48.9499,B 2.3914,C 0.2556,E1 2.5,E2 502.0342} C_DIS
LIN {X 74.907,Y -112.0859,Z 188,A -50.5989,B 2.3912,C 0.2583,E1 2.4962,E2 503.6815} C_DIS
LIN {X 71.4659,Y -114.311,Z 188,A -52.0844,B 2.391,C 0.2593,E1 2.4928,E2 505.1348} C_DIS
LIN {X 68.4722,Y -116.1288,Z 188,A -53.8463,B 2.3906,C 0.2637,E1 2.4884,E2 506.9335} C_DIS
LIN {X 64.3787,Y -118.4472,Z 188,A -55.6609,B 2.3904,C 0.2654,E1 2.4841,E2 508.7255} C_DIS
LIN {X 60.87,Y -120.2859,Z 188,A -57.149,B 2.3903,C 0.2664,E1 2.4804,E2 510.1891} C_DIS
LIN {X 57.9917,Y -121.6994,Z 188,A -58.5611,B 2.39,C 0.2686,E1 2.4768,E2 511.6086} C_DIS
LIN {X 50.2662,Y -125.0884,Z 188,A -61.9921,B 2.3896,C 0.2722,E1 2.4681,E2 515.0218} C_DIS
LIN {X 46.5922,Y -126.5049,Z 188,A -63.9865,B 2.3891,C 0.2763,E1 2.4627,E2 517.0595} C_DIS
LIN {X 43.0917,Y -127.7387,Z 188,A -65.029,B 2.3894,C 0.2744,E1 2.4602,E2 518.0327} C_DIS
LIN {X 38.8814,Y -129.0829,Z 188,A -66.9326,B 2.3891,C 0.2765,E1 2.4551,E2 519.941} C_DIS
LIN {X 36.1819,Y -129.8642,Z 188,A -68.127,B 2.389,C 0.2776,E1 2.4518,E2 521.136} C_DIS
LIN {X 33.2726,Y -130.6398,Z 188,A -69.5288,B 2.3888,C 0.2796,E1 2.448,E2 522.5548} C_DIS
LIN {X 29.2859,Y -131.5931,Z 188,A -71.1016,B 2.3888,C 0.2799,E1 2.4438,E2 524.1064} C_DIS
LIN {X 26.7895,Y -132.1218,Z 188,A -72.2755,B 2.3886,C 0.2813,E1 2.4405,E2 525.2926} C_DIS
LIN {X 23.1533,Y -132.8086,Z 188,A -73.6952,B 2.3886,C 0.2815,E1 2.4367,E2 526.6931} C_DIS
LIN {X 19.7649,Y -133.3555,Z 188,A -75.1269,B 2.3885,C 0.2822,E1 2.4327,E2 528.1222} C_DIS
LIN {X 16.5529,Y -133.7917,Z 188,A -76.7999,B 2.3882,C 0.2848,E1 2.428,E2 529.8348} C_DIS
LIN {X 12.5178,Y -134.2286,Z 188,A -78.2879,B 2.3882,C 0.2842,E1 2.4239,E2 531.2925} C_DIS
LIN {X 9.3425,Y -134.4873,Z 188,A -79.568,B 2.3882,C 0.2842,E1 2.4204,E2 532.5636} C_DIS
LIN {X 4.3093,Y -134.7429,Z 188,A -82.1399,B 2.3878,C 0.2875,E1 2.413,E2 535.1932} C_DIS
LIN {X 0.9849,Y -134.8006,Z 188,A -82.3039,B 2.3886,C 0.2806,E1 2.413,E2 535.1923} C_DIS
Enddeposition()
LIN {X 0.9849,Y -134.8006,Z 188,A -82.3042,B 2.3886,C 0.2806,E1 2.413,E2 535.1927} C_DIS
Startdeposition()
$VEL.CP = VEL_PRINT
LIN {X 2.0471,Y -135.6947,Z 188,A -81.2221,B 2.389,C 0.278,E1 2.4162,E2 534.0541} C_DIS
LIN {X 8.0811,Y -135.4694,Z 188,A -79.4747,B 2.3885,C 0.2819,E1 2.4208,E2 532.4139} C_DIS
LIN {X 16.3306,Y -134.7239,Z 188,A -76.0206,B 2.3887,C 0.2805,E1 2.4304,E2 528.9638} C_DIS
LIN {X 22.4824,Y -133.8346,Z 188,A -73.4338,B 2.3888,C 0.2791,E1 2.4376,E2 526.3806} C_DIS
LIN {X 26.4089,Y -133.117,Z 188,A -71.6894,B 2.389,C 0.2775,E1 2.4424,E2 524.6274} C_DIS
LIN {X 31.3728,Y -132.0343,Z 188,A -69.622,B 2.3892,C 0.2763,E1 2.448,E2 522.5691} C_DIS
LIN {X 34.6951,Y -131.2,Z 188,A -68.237,B 2.3892,C 0.2754,E1 2.4517,E2 521.1914} C_DIS
LIN {X 37.6821,Y -130.374,Z 188,A -67.046,B 2.3893,C 0.2749,E1 2.4549,E2 520.0152} C_DIS
LIN {X 41.1458,Y -129.3218,Z 188,A -65.5326,B 2.3895,C 0.2735,E1 2.4589,E2 518.5029} C_DIS
LIN {X 44.8324,Y -128.0909,Z 188,A -63.7047,B 2.3898,C 0.2704,E1 2.4638,E2 516.6488} C_DIS
LIN {X 48.3449,Y -126.8088,Z 188,A -62.3348,B 2.3898,C 0.2701,E1 2.4674,E2 515.306} C_DIS
LIN {X 55.8354,Y -123.6918,Z 188,A -58.9832,B 2.3903,C 0.2663,E1 2.476,E2 511.962} C_DIS
LIN {X 59.6195,Y -121.913,Z 188,A -57.2444,B 2.3906,C 0.264,E1 2.4804,E2 510.2255} C_DIS
LIN {X 62.4962,Y -120.4646,Z 188,A -55.8418,B 2.3908,C 0.2618,E1 2.4839,E2 508.8162} C_DIS
LIN {X 65.4486,Y -118.8873,Z 188,A -53.7673,B 2.3916,C 0.2548,E1 2.4892,E2 506.6518} C_DIS
LIN {X 70.8265,Y -115.7637,Z 188,A -51.9767,B 2.3913,C 0.2568,E1 2.4932,E2 504.9716} C_DIS
LIN {X 74.3472,Y -113.535,Z 188,A -50.2745,B 2.3916,C 0.2543,E1 2.4972,E2 503.2757} C_DIS
LIN {X 77.4085,Y -111.4699,Z 188,A -48.6362,B 2.392,C 0.251,E1 2.501,E2 501.6256} C_DIS
LIN {X 82.6153,Y -107.6678,Z 188,A -46.1412,B 2.3923,C 0.2478,E1 2.5065,E2 499.1589} C_DIS
LIN {X 85.8937,Y -105.0707,Z 188,A -43.9023,B 2.393,C 0.2408,E1 2.5115,E2 496.8554} C_DIS
LIN {X 89.8079,Y -101.7454,Z 188,A -42.267,B 2.393,C 0.2408,E1 2.5148,E2 495.2897} C_DIS
LIN {X 93.5395,Y -98.3262,Z 188,A -40.2693,B 2.3933,C 0.2375,E1 2.5188,E2 493.3089} C_DIS
LIN {X 96.7467,Y -95.1719,Z 188,A -37.9709,B 2.394,C 0.2303,E1 2.5235,E2 490.9558} C_DIS
LIN {X 100.2072,Y -91.5214,Z 188,A -36.4238,B 2.394,C 0.2303,E1 2.5262,E2 489.4838} C_DIS
LIN {X 104.496,Y -86.5921,Z 188,A -33.8005,B 2.3945,C 0.2253,E1 2.531,E2 486.8762} C_DIS
LIN {X 108.7508,Y -81.184,Z 188,A -30.8791,B 2.3951,C 0.2185,E1 2.536,E2 483.9504} C_DIS
LIN {X 113.1141,Y -74.9864,Z 188,A -27.963,B 2.3956,C 0.2132,E1 2.5405,E2 481.0693} C_DIS
LIN {X 115.3664,Y -71.4721,Z 188,A -26.4112,B 2.3959,C 0.2106,E1 2.5428,E2 479.5439} C_DIS
LIN {X 117.5999,Y -67.7344,Z 188,A -24.5421,B 2.3963,C 0.2058,E1 2.5455,E2 477.6692} C_DIS
LIN {X 119.8003,Y -63.761,Z 188,A -22.736,B 2.3966,C 0.2019,E1 2.5478,E2 475.8763} C_DIS
LIN {X 121.4258,Y -60.6071,Z 188,A -21.3593,B 2.3968,C 0.1991,E1 2.5496,E2 474.5143} C_DIS
LIN {X 122.9679,Y -57.4124,Z 188,A -19.909,B 2.3971,C 0.1957,E1 2.5513,E2 473.069} C_DIS
LIN {X 124.4849,Y -54.0425,Z 188,A -17.812,B 2.3978,C 0.1871,E1 2.5537,E2 470.9004} C_DIS
LIN {X 126.6352,Y -48.7928,Z 188,A -16.1454,B 2.3978,C 0.1869,E1 2.5553,E2 469.3275} C_DIS
LIN {X 129.4614,Y -40.7089,Z 188,A -12.6753,B 2.3985,C 0.1784,E1 2.5584,E2 465.8739} C_DIS
LIN {X 130.5384,Y -37.11,Z 188,A -11.2268,B 2.3987,C 0.1753,E1 2.5595,E2 464.442} C_DIS
LIN {X 131.4664,Y -33.6717,Z 188,A -9.8989,B 2.3989,C 0.1726,E1 2.5604,E2 463.1357} C_DIS
LIN {X 132.2693,Y -30.3639,Z 188,A -8.5508,B 2.3991,C 0.1694,E1 2.5613,E2 461.798} C_DIS
LIN {X 133.0272,Y -26.8501,Z 188,A -7.078,B 2.3994,C 0.1656,E1 2.5621,E2 460.3301} C_DIS
LIN {X 133.8016,Y -22.6804,Z 188,A -5.3975,B 2.3997,C 0.1616,E1 2.563,E2 458.6625} C_DIS
LIN {X 134.601,Y -17.3154,Z 188,A -3.2572,B 2.4,C 0.1565,E1 2.5638,E2 456.5398} C_DIS
LIN {X 134.904,Y -14.7695,Z 188,A -1.8725,B 2.4004,C 0.1509,E1 2.5642,E2 455.1156} C_DIS
LIN {X 135.2568,Y -11.085,Z 188,A -0.6381,B 2.4004,C 0.1493,E1 2.5645,E2 453.9224} C_DIS
LIN {X 135.5588,Y -6.415,Z 188,A 1.1949,B 2.4007,C 0.1449,E1 2.5648,E2 452.1064} C_DIS
LIN {X 135.6634,Y -3.5613,Z 188,A 2.4743,B 2.401,C 0.1409,E1 2.5648,E2 450.8168} C_DIS
LIN {X 135.6525,Y 3.9553,Z 188,A 5.3537,B 2.4013,C 0.1345,E1 2.5648,E2 447.973} C_DIS
LIN {X 135.4336,Y 8.6613,Z 188,A 7.6741,B 2.4018,C 0.1261,E1 2.5644,E2 445.6092} C_DIS
LIN {X 135.043,Y 13.4455,Z 188,A 9.3616,B 2.4019,C 0.1233,E1 2.564,E2 443.9639} C_DIS
LIN {X 134.6465,Y 16.9684,Z 188,A 10.5367,B 2.402,C 0.1218,E1 2.5636,E2 442.8288} C_DIS
LIN {X 134.0147,Y 21.3919,Z 188,A 12.4375,B 2.4023,C 0.1165,E1 2.5628,E2 440.9252} C_DIS
LIN {X 133.2738,Y 25.5974,Z 188,A 13.958,B 2.4023,C 0.1138,E1 2.562,E2 439.4393} C_DIS
LIN {X 132.4483,Y 29.5802,Z 188,A 15.5023,B 2.4025,C 0.1106,E1 2.5611,E2 437.916} C_DIS
LIN {X 131.6117,Y 33.0989,Z 188,A 16.9491,B 2.4027,C 0.107,E1 2.5602,E2 436.4784} C_DIS
LIN {X 130.7835,Y 36.2337,Z 188,A 18.336,B 2.4029,C 0.1032,E1 2.5592,E2 435.0886} C_DIS
LIN {X 129.735,Y 39.8237,Z 188,A 19.798,B 2.403,C 0.0999,E1 2.558,E2 433.6405} C_DIS
LIN {X 128.6568,Y 43.1812,Z 188,A 21.2629,B 2.4032,C 0.0961,E1 2.5567,E2 432.1779} C_DIS
LIN {X 127.4507,Y 46.6238,Z 188,A 22.8318,B 2.4033,C 0.0917,E1 2.5552,E2 430.6049} C_DIS
LIN {X 125.4924,Y 51.6638,Z 188,A 24.8335,B 2.4035,C 0.088,E1 2.5532,E2 428.6373} C_DIS
LIN {X 124.1523,Y 54.8059,Z 188,A 26.1813,B 2.4035,C 0.085,E1 2.5517,E2 427.3007} C_DIS
LIN {X 122.2703,Y 58.883,Z 188,A 28.0976,B 2.4038,C 0.08,E1 2.5494,E2 425.3811} C_DIS
LIN {X 120.3293,Y 62.7538,Z 188,A 29.6854,B 2.4038,C 0.0773,E1 2.5474,E2 423.8225} C_DIS
LIN {X 118.468,Y 66.2045,Z 188,A 31.3203,B 2.404,C 0.0733,E1 2.5453,E2 422.1897} C_DIS
LIN {X 115.3604,Y 71.4817,Z 188,A 33.7038,B 2.4041,C 0.0686,E1 2.5419,E2 419.8303} C_DIS
LIN {X 111.6731,Y 77.1159,Z 188,A 36.5687,B 2.4043,C 0.0616,E1 2.5374,E2 416.9621} C_DIS
LIN {X 109.2091,Y 80.567,Z 188,A 38.2631,B 2.4043,C 0.0582,E1 2.5347,E2 415.279} C_DIS
LIN {X 106.6054,Y 83.9816,Z 188,A 39.9522,B 2.4045,C 0.055,E1 2.5318,E2 413.6048} C_DIS
LIN {X 103.9992,Y 87.1881,Z 188,A 41.6313,B 2.4045,C 0.0516,E1 2.5288,E2 411.9333} C_DIS
LIN {X 101.2512,Y 90.365,Z 188,A 43.3522,B 2.4046,C 0.0481,E1 2.5257,E2 410.2185} C_DIS
LIN {X 98.9879,Y 92.8393,Z 188,A 45.1988,B 2.4047,C 0.0419,E1 2.522,E2 408.3189} C_DIS
LIN {X 95.5883,Y 96.3352,Z 188,A 46.4251,B 2.4047,C 0.0439,E1 2.5198,E2 407.1942} C_DIS
LIN {X 90.0421,Y 101.5384,Z 188,A 49.7779,B 2.4048,C 0.0364,E1 2.5129,E2 403.824} C_DIS
LIN {X 86.6877,Y 104.4167,Z 188,A 51.562,B 2.4048,C 0.0334,E1 2.5091,E2 402.0498} C_DIS
LIN {X 83.4073,Y 107.0557,Z 188,A 53.28,B 2.4048,C 0.0306,E1 2.5054,E2 400.339} C_DIS
LIN {X 79.9001,Y 109.6981,Z 188,A 55.0957,B 2.4049,C 0.0276,E1 2.5013,E2 398.5278} C_DIS
LIN {X 76.0386,Y 112.4087,Z 188,A 56.9318,B 2.4049,C 0.0253,E1 2.4971,E2 396.7106} C_DIS
LIN {X 70.7549,Y 115.8076,Z 188,A 59.2552,B 2.4049,C 0.0232,E1 2.4917,E2 394.427} C_DIS
LIN {X 64.8096,Y 119.2365,Z 188,A 62.3839,B 2.405,C 0.0173,E1 2.4841,E2 391.2709} C_DIS
LIN {X 61.3428,Y 121.0544,Z 188,A 63.8426,B 2.405,C 0.0162,E1 2.4805,E2 389.8356} C_DIS
LIN {X 57.7882,Y 122.7933,Z 188,A 65.9623,B 2.405,C 0.0111,E1 2.475,E2 387.6622} C_DIS
LIN {X 54.0259,Y 124.4921,Z 188,A 67.1614,B 2.405,C 0.0124,E1 2.4721,E2 386.5286} C_DIS
LIN {X 51.0842,Y 125.7283,Z 188,A 68.6091,B 2.405,C 0.0101,E1 2.4683,E2 385.0691} C_DIS
LIN {X 48.1735,Y 126.873,Z 188,A 69.7772,B 2.405,C 0.0095,E1 2.4653,E2 383.9195} C_DIS
LIN {X 44.8809,Y 128.0741,Z 188,A 71.3691,B 2.405,C 0.0072,E1 2.4611,E2 382.3144} C_DIS
LIN {X 40.2785,Y 129.5958,Z 188,A 73.2304,B 2.405,C 0.0063,E1 2.4562,E2 380.4758} C_DIS
LIN {X 36.9648,Y 130.579,Z 188,A 74.7434,B 2.405,C 0.0046,E1 2.4521,E2 378.9567} C_DIS
LIN {X 33.7727,Y 131.4407,Z 188,A 75.9848,B 2.405,C 0.0043,E1 2.4488,E2 377.734} C_DIS
LIN {X 30.2558,Y 132.294,Z 188,A 77.5563,B 2.405,C 0.0028,E1 2.4445,E2 376.1577} C_DIS
LIN {X 26.7226,Y 133.0532,Z 188,A 79.1506,B 2.405,C 0.0013,E1 2.4401,E2 374.5558} C_DIS
LIN {X 22.6408,Y 133.8082,Z 188,A 81.025,B 2.405,C -0.0005,E1 2.4349,E2 372.6673} C_DIS
LIN {X 17.8808,Y 134.5269,Z 188,A 82.8023,B 2.405,C -0.0002,E1 2.4301,E2 370.9211} C_DIS
LIN {X 14.3591,Y 134.9481,Z 188,A 84.3289,B 2.405,C -0.0011,E1 2.4258,E2 369.3916} C_DIS
LIN {X 11.2612,Y 135.2419,Z 188,A 85.866,B 2.405,C -0.0028,E1 2.4215,E2 367.8284} C_DIS
LIN {X 7.9407,Y 135.478,Z 188,A 87.4601,B 2.405,C -0.0043,E1 2.4169,E2 366.2123} C_DIS
LIN {X 3.6294,Y 135.6615,Z 188,A 88.7743,B 2.405,C -0.0021,E1 2.4134,E2 364.9593} C_DIS
LIN {X -0.0141,Y 135.712,Z 188,A 90.2896,B 2.405,C -0.0022,E1 2.4092,E2 363.4475} C_DIS
LIN {X -3.5347,Y 135.6641,Z 188,A 92.0523,B 2.405,C -0.0038,E1 2.4042,E2 361.6525} C_DIS
LIN {X -10.5921,Y 135.2978,Z 188,A 94.8075,B 2.405,C -0.0027,E1 2.3966,E2 358.9259} C_DIS
LIN {X -14.0479,Y 134.9816,Z 188,A 96.229,B 2.405,C -0.0023,E1 2.3926,E2 357.5102} C_DIS
LIN {X -19.6758,Y 134.2767,Z 188,A 98.7714,B 2.405,C -0.0025,E1 2.3855,E2 354.9514} C_DIS
LIN {X -23.6801,Y 133.628,Z 188,A 100.3617,B 2.405,C -0.0014,E1 2.3812,E2 353.3766} C_DIS
LIN {X -26.4639,Y 133.1058,Z 188,A 101.6771,B 2.405,C -0.0015,E1 2.3775,E2 352.0476} C_DIS
LIN {X -29.8641,Y 132.3835,Z 188,A 103.1004,B 2.405,C -0.0007,E1 2.3737,E2 350.6303} C_DIS
LIN {X -32.7436,Y 131.7019,Z 188,A 104.3833,B 2.405,C -0.0002,E1 2.3702,E2 349.3442} C_DIS
LIN {X -36.3819,Y 130.7421,Z 188,A 105.9643,B 2.405,C 0.0008,E1 2.3659,E2 347.7649} C_DIS
LIN {X -39.6891,Y 129.7762,Z 188,A 107.2828,B 2.405,C 0.0023,E1 2.3624,E2 346.4633} C_DIS
LIN {X -42.2378,Y 128.9709,Z 188,A 109.2305,B 2.405,C -0.0003,E1 2.357,E2 344.4187} C_DIS
LIN {X -47.1383,Y 127.2607,Z 188,A 110.6446,B 2.405,C 0.0046,E1 2.3535,E2 343.0987} C_DIS
LIN {X -50.4778,Y 125.9727,Z 188,A 112.4102,B 2.405,C 0.0049,E1 2.3488,E2 341.3038} C_DIS
LIN {X -54.0068,Y 124.5004,Z 188,A 113.8236,B 2.405,C 0.0073,E1 2.3452,E2 339.9153} C_DIS
LIN {X -56.3647,Y 123.4524,Z 188,A 115.2311,B 2.405,C 0.0072,E1 2.3416,E2 338.4707} C_DIS
LIN {X -60.0697,Y 121.6909,Z 188,A 116.8046,B 2.405,C 0.0096,E1 2.3377,E2 336.917} C_DIS
LIN {X -62.9207,Y 120.2416,Z 188,A 118.02,B 2.405,C 0.0117,E1 2.3347,E2 335.7185} C_DIS
LIN {X -68.8701,Y 116.9381,Z 188,A 120.9554,B 2.405,C 0.0151,E1 2.3275,E2 332.7779} C_DIS
LIN {X -74.0173,Y 113.7499,Z 188,A 123.8617,B 2.405,C 0.0173,E1 2.3205,E2 329.8318} C_DIS
LIN {X -77.4539,Y 111.4383,Z 188,A 125.6876,B 2.405,C 0.0196,E1 2.3163,E2 327.9978} C_DIS
LIN {X -83.8451,Y 106.7127,Z 188,A 129.2123,B 2.405,C 0.0244,E1 2.3084,E2 324.4553} C_DIS
LIN {X -87.2363,Y 103.9587,Z 188,A 131.0749,B 2.405,C 0.0274,E1 2.3043,E2 322.5919} C_DIS
LIN {X -90.1711,Y 101.4244,Z 188,A 132.9603,B 2.405,C 0.0296,E1 2.3003,E2 320.6778} C_DIS
LIN {X -92.6356,Y 99.178,Z 188,A 134.7474,B 2.4049,C 0.031,E1 2.2966,E2 318.8458} C_DIS
LIN {X -95.9329,Y 95.9928,Z 188,A 136.2749,B 2.4049,C 0.0359,E1 2.2937,E2 317.3691} C_DIS
LIN {X -98.9706,Y 92.8577,Z 188,A 137.9615,B 2.4048,C 0.0399,E1 2.2904,E2 315.7026} C_DIS
LIN {X -102.6109,Y 88.8183,Z 188,A 140.8826,B 2.4048,C 0.0428,E1 2.2849,E2 312.7078} C_DIS
LIN {X -104.8765,Y 86.1314,Z 188,A 142.1829,B 2.4046,C 0.0464,E1 2.2826,E2 311.4307} C_DIS
LIN {X -107.3756,Y 82.9946,Z 188,A 143.8727,B 2.4046,C 0.0501,E1 2.2797,E2 309.7426} C_DIS
LIN {X -109.9506,Y 79.5516,Z 188,A 145.8365,B 2.4045,C 0.0537,E1 2.2764,E2 307.7622} C_DIS
LIN {X -112.564,Y 75.8093,Z 188,A 147.7998,B 2.4044,C 0.058,E1 2.2733,E2 305.7959} C_DIS
LIN {X -114.882,Y 72.2479,Z 188,A 149.7782,B 2.4043,C 0.0617,E1 2.2703,E2 303.7963} C_DIS
LIN {X -117.736,Y 67.4975,Z 188,A 152.2715,B 2.4042,C 0.0669,E1 2.2667,E2 301.286} C_DIS
LIN {X -119.8854,Y 63.5991,Z 188,A 154.2714,B 2.404,C 0.0711,E1 2.2641,E2 299.2727} C_DIS
LIN {X -121.6346,Y 60.1837,Z 188,A 155.8236,B 2.404,C 0.0753,E1 2.2621,E2 297.7299} C_DIS
LIN {X -123.0927,Y 57.1427,Z 188,A 157.3438,B 2.4038,C 0.0787,E1 2.2603,E2 296.199} C_DIS
LIN {X -124.6894,Y 53.5695,Z 188,A 159.1348,B 2.4037,C 0.0826,E1 2.2583,E2 294.3923} C_DIS
LIN {X -126.3586,Y 49.5045,Z 188,A 161.0175,B 2.4035,C 0.0873,E1 2.2563,E2 292.5075} C_DIS
LIN {X -127.5797,Y 46.2662,Z 188,A 162.628,B 2.4034,C 0.0908,E1 2.2547,E2 290.8796} C_DIS
LIN {X -128.6237,Y 43.2805,Z 188,A 164.0312,B 2.4032,C 0.0942,E1 2.2535,E2 289.4691} C_DIS
LIN {X -129.8376,Y 39.4884,Z 188,A 165.839,B 2.4031,C 0.0984,E1 2.2519,E2 287.6468} C_DIS
LIN {X -131.0093,Y 35.4102,Z 188,A 167.7335,B 2.4029,C 0.103,E1 2.2505,E2 285.7408} C_DIS
LIN {X -132.339,Y 30.0588,Z 188,A 170.3165,B 2.4026,C 0.1088,E1 2.2488,E2 283.1277} C_DIS
LIN {X -133.2451,Y 25.7479,Z 188,A 171.971,B 2.4024,C 0.1144,E1 2.2479,E2 281.5} C_DIS
LIN {X -133.8204,Y 22.5673,Z 188,A 173.6655,B 2.4022,C 0.1174,E1 2.2471,E2 279.7654} C_DIS
LIN {X -134.4578,Y 18.4082,Z 188,A 175.5926,B 2.402,C 0.122,E1 2.2463,E2 277.8207} C_DIS
LIN {X -134.9236,Y 14.5873,Z 188,A 177.1318,B 2.4017,C 0.1268,E1 2.2458,E2 276.2932} C_DIS
LIN {X -135.2125,Y 11.6101,Z 188,A 178.5986,B 2.4016,C 0.1299,E1 2.2454,E2 274.8017} C_DIS
LIN {X -135.5042,Y 7.5023,Z 188,A -179.514,B 2.4013,C 0.1344,E1 2.2451,E2 272.8968} C_DIS
LIN {X -135.6562,Y 3.8197,Z 188,A -177.89,B 2.4011,C 0.1386,E1 2.2449,E2 271.2652} C_DIS
LIN {X -135.7112,Y -0.3631,Z 188,A -175.9543,B 2.4008,C 0.1432,E1 2.2449,E2 269.3093} C_DIS
LIN {X -135.6333,Y -4.6096,Z 188,A -174.0173,B 2.4005,C 0.148,E1 2.2451,E2 267.3551} C_DIS
LIN {X -135.4527,Y -8.3522,Z 188,A -172.48,B 2.4003,C 0.1525,E1 2.2453,E2 265.8244} C_DIS
LIN {X -135.1845,Y -11.9415,Z 188,A -170.7468,B 2.4,C 0.1563,E1 2.2457,E2 264.065} C_DIS
LIN {X -134.7481,Y -16.1278,Z 188,A -168.9612,B 2.3997,C 0.1612,E1 2.2463,E2 262.2793} C_DIS
LIN {X -134.2708,Y -19.7176,Z 188,A -167.2211,B 2.3994,C 0.165,E1 2.2469,E2 260.5131} C_DIS
LIN {X -133.628,Y -23.6801,Z 188,A -165.6236,B 2.3991,C 0.1699,E1 2.2477,E2 258.929} C_DIS
LIN {X -133.0517,Y -26.7299,Z 188,A -164.1571,B 2.3989,C 0.1731,E1 2.2485,E2 257.4433} C_DIS
LIN {X -132.2777,Y -30.3272,Z 188,A -162.4535,B 2.3986,C 0.177,E1 2.2495,E2 255.7212} C_DIS
LIN {X -131.2545,Y -34.4904,Z 188,A -160.4337,B 2.3982,C 0.1814,E1 2.2509,E2 253.6754} C_DIS
LIN {X -130.1201,Y -38.5491,Z 188,A -158.4894,B 2.3979,C 0.1858,E1 2.2525,E2 251.7107} C_DIS
LIN {X -128.0874,Y -44.8426,Z 188,A -155.8417,B 2.3973,C 0.1935,E1 2.2548,E2 249.0828} C_DIS
LIN {X -126.765,Y -48.459,Z 188,A -153.9,B 2.397,C 0.1969,E1 2.2567,E2 247.1012} C_DIS
LIN {X -125.4505,Y -51.7646,Z 188,A -152.3154,B 2.3967,C 0.2006,E1 2.2584,E2 245.5064} C_DIS
LIN {X -123.997,Y -55.1532,Z 188,A -150.8008,B 2.3964,C 0.2046,E1 2.2601,E2 243.9979} C_DIS
LIN {X -122.6051,Y -58.182,Z 188,A -149.2182,B 2.3961,C 0.2077,E1 2.262,E2 242.3931} C_DIS
LIN {X -121.014,Y -61.422,Z 188,A -147.7084,B 2.3958,C 0.2115,E1 2.2639,E2 240.8857} C_DIS
LIN {X -118.6427,Y -65.8904,Z 188,A -145.4343,B 2.3954,C 0.2163,E1 2.2669,E2 238.5944} C_DIS
LIN {X -116.728,Y -69.2261,Z 188,A -143.7557,B 2.395,C 0.2199,E1 2.2693,E2 236.9092} C_DIS
LIN {X -114.9781,Y -72.0955,Z 188,A -142.2047,B 2.3947,C 0.2229,E1 2.2716,E2 235.3414} C_DIS
LIN {X -112.7653,Y -75.509,Z 188,A -140.3337,B 2.3944,C 0.2263,E1 2.2745,E2 233.4508} C_DIS
LIN {X -110.1634,Y -79.2576,Z 188,A -138.2796,B 2.3941,C 0.2302,E1 2.2778,E2 231.3805} C_DIS
LIN {X -107.5008,Y -82.833,Z 188,A -136.3278,B 2.3937,C 0.234,E1 2.2811,E2 229.4199} C_DIS
LIN {X -104.7378,Y -86.3,Z 188,A -134.3326,B 2.3933,C 0.2375,E1 2.2847,E2 227.4088} C_DIS
LIN {X -101.4717,Y -90.1175,Z 188,A -132.4486,B 2.3928,C 0.2426,E1 2.2881,E2 225.5563} C_DIS
LIN {X -98.444,Y -93.4159,Z 188,A -130.1419,B 2.3926,C 0.2449,E1 2.2926,E2 223.1951} C_DIS
LIN {X -95.4664,Y -96.4563,Z 188,A -128.1981,B 2.3923,C 0.2478,E1 2.2964,E2 221.2321} C_DIS
LIN {X -91.7552,Y -99.9929,Z 188,A -126.0942,B 2.3919,C 0.2519,E1 2.3007,E2 219.1364} C_DIS
LIN {X -88.4156,Y -102.9578,Z 188,A -124.1595,B 2.3915,C 0.2549,E1 2.3048,E2 217.1953} C_DIS
LIN {X -85.1197,Y -105.6988,Z 188,A -122.2686,B 2.3913,C 0.2576,E1 2.3089,E2 215.2938} C_DIS
LIN {X -81.7115,Y -108.3551,Z 188,A -120.4048,B 2.391,C 0.2603,E1 2.3131,E2 213.4247} C_DIS
LIN {X -78.2296,Y -110.8951,Z 188,A -118.0946,B 2.3909,C 0.2611,E1 2.3185,E2 211.049} C_DIS
LIN {X -74.8114,Y -113.2294,Z 188,A -116.7042,B 2.3905,C 0.265,E1 2.3216,E2 209.7063} C_DIS
LIN {X -71.4283,Y -115.3936,Z 188,A -115.1798,B 2.3901,C 0.268,E1 2.3252,E2 208.2046} C_DIS
LIN {X -68.1644,Y -117.351,Z 188,A -113.2518,B 2.3901,C 0.2687,E1 2.3299,E2 206.2337} C_DIS
LIN {X -64.0183,Y -119.6633,Z 188,A -111.1491,B 2.3898,C 0.2706,E1 2.3351,E2 204.1177} C_DIS
LIN {X -60.616,Y -121.4214,Z 188,A -109.2181,B 2.3898,C 0.271,E1 2.34,E2 202.1442} C_DIS
LIN {X -57.1203,Y -123.103,Z 188,A -107.9806,B 2.3894,C 0.2744,E1 2.343,E2 200.9601} C_DIS
LIN {X -53.9721,Y -124.5154,Z 188,A -106.4996,B 2.3892,C 0.2757,E1 2.3468,E2 199.4757} C_DIS
LIN {X -50.7607,Y -125.8587,Z 188,A -105.0102,B 2.3892,C 0.2769,E1 2.3507,E2 197.9833} C_DIS
LIN {X -47.9411,Y -126.96,Z 188,A -103.5818,B 2.3891,C 0.2773,E1 2.3545,E2 196.5345} C_DIS
LIN {X -43.5776,Y -128.5248,Z 188,A -101.6026,B 2.3889,C 0.2786,E1 2.3597,E2 194.5519} C_DIS
LIN {X -39.9376,Y -129.7002,Z 188,A -100.0846,B 2.3887,C 0.2801,E1 2.3637,E2 193.0464} C_DIS
LIN {X -36.9175,Y -130.5923,Z 188,A -98.8139,B 2.3887,C 0.2812,E1 2.3671,E2 191.7832} C_DIS
LIN {X -33.4362,Y -131.5261,Z 188,A -97.1842,B 2.3886,C 0.2814,E1 2.3716,E2 190.1386} C_DIS
LIN {X -29.9598,Y -132.3616,Z 188,A -95.6125,B 2.3886,C 0.2818,E1 2.3759,E2 188.5581} C_DIS
LIN {X -25.6436,Y -133.265,Z 188,A -94.022,B 2.3883,C 0.2839,E1 2.3802,E2 187.0034} C_DIS
LIN {X -21.5819,Y -133.9848,Z 188,A -91.8842,B 2.3885,C 0.2822,E1 2.3862,E2 184.8118} C_DIS
LIN {X -17.3503,Y -134.5964,Z 188,A -90.2146,B 2.3884,C 0.2833,E1 2.3908,E2 183.1596} C_DIS
LIN {X -14.1823,Y -134.9672,Z 188,A -88.7742,B 2.3884,C 0.2829,E1 2.3948,E2 181.7062} C_DIS
LIN {X -6.1913,Y -135.5701,Z 188,A -85.4857,B 2.3884,C 0.2834,E1 2.404,E2 178.4291} C_DIS
LIN {X 0.9946,Y -135.706,Z 188,A -82.6087,B 2.3883,C 0.2838,E1 2.412,E2 175.5719} C_DIS
Enddeposition()
LIN {X 0.9946,Y -135.706,Z 188,A -82.6088,B 2.3883,C 0.2838,E1 2.412,E2 175.572} C_DIS
Startdeposition()
$VEL.CP = VEL_PRINT
LIN {X -0.2215,Y -136.6102,Z 188,A -84.1059,B 2.2797,C 0.2862,E1 2.2995,E2 177.262} C_DIS
LIN {X -5.7865,Y -136.4875,Z 188,A -85.5566,B 2.2802,C 0.2817,E1 2.2957,E2 178.5954} C_DIS
LIN {X -10.1386,Y -136.2326,Z 188,A -87.8214,B 2.2799,C 0.284,E1 2.2892,E2 180.9197} C_DIS
LIN {X -15.2159,Y -135.7605,Z 188,A -90.0132,B 2.2799,C 0.2841,E1 2.2831,E2 183.1196} C_DIS
LIN {X -18.6634,Y -135.3299,Z 188,A -91.2063,B 2.2801,C 0.2826,E1 2.2799,E2 184.2778} C_DIS
LIN {X -23.1468,Y -134.635,Z 188,A -93.225,B 2.2801,C 0.2826,E1 2.2743,E2 186.3127} C_DIS
LIN {X -27.3442,Y -133.8444,Z 188,A -94.8289,B 2.2803,C 0.2812,E1 2.2699,E2 187.892} C_DIS
LIN {X -30.8289,Y -133.0856,Z 188,A -96.3194,B 2.2803,C 0.2805,E1 2.2659,E2 189.3824} C_DIS
LIN {X -33.8849,Y -132.3401,Z 188,A -97.7041,B 2.2803,C 0.2802,E1 2.2621,E2 190.7763} C_DIS
LIN {X -37.4234,Y -131.3846,Z 188,A -99.2347,B 2.2805,C 0.2794,E1 2.2579,E2 192.3064} C_DIS
LIN {X -40.4351,Y -130.4884,Z 188,A -100.5779,B 2.2805,C 0.2787,E1 2.2543,E2 193.6535} C_DIS
LIN {X -43.7162,Y -129.4265,Z 188,A -102.0766,B 2.2807,C 0.2779,E1 2.2503,E2 195.1595} C_DIS
LIN {X -48.2974,Y -127.7869,Z 188,A -104.1649,B 2.2808,C 0.2766,E1 2.2448,E2 197.2546} C_DIS
LIN {X -51.2327,Y -126.6381,Z 188,A -105.5153,B 2.281,C 0.2756,E1 2.2413,E2 198.6091} C_DIS
LIN {X -54.6626,Y -125.1966,Z 188,A -107.102,B 2.2811,C 0.2743,E1 2.2372,E2 200.1996} C_DIS
LIN {X -59.3008,Y -123.0673,Z 188,A -109.4444,B 2.2813,C 0.2729,E1 2.2312,E2 202.5693} C_DIS
LIN {X -62.8192,Y -121.3107,Z 188,A -111.1004,B 2.2815,C 0.2712,E1 2.2271,E2 204.2266} C_DIS
LIN {X -66.9708,Y -119.0689,Z 188,A -113.0937,B 2.2818,C 0.2689,E1 2.2222,E2 206.2219} C_DIS
LIN {X -73.8765,Y -114.9123,Z 188,A -117.2932,B 2.2819,C 0.2675,E1 2.212,E2 210.5301} C_DIS
LIN {X -78.7902,Y -111.6002,Z 188,A -119.0939,B 2.2826,C 0.2615,E1 2.208,E2 212.2404} C_DIS
LIN {X -82.0263,Y -109.2442,Z 188,A -120.9232,B 2.2829,C 0.2594,E1 2.2039,E2 214.0897} C_DIS
LIN {X -85.661,Y -106.4176,Z 188,A -122.8917,B 2.2832,C 0.2565,E1 2.1995,E2 216.0631} C_DIS
LIN {X -89.2143,Y -103.4568,Z 188,A -124.9088,B 2.2835,C 0.2535,E1 2.1952,E2 218.0903} C_DIS
LIN {X -92.5746,Y -100.4613,Z 188,A -126.8586,B 2.2839,C 0.2504,E1 2.1911,E2 220.0481} C_DIS
LIN {X -95.9641,Y -97.229,Z 188,A -128.8359,B 2.2842,C 0.2468,E1 2.1872,E2 222.0269} C_DIS
LIN {X -98.3775,Y -94.7865,Z 188,A -130.6089,B 2.2844,C 0.2451,E1 2.1836,E2 223.8436} C_DIS
LIN {X -102.3331,Y -90.501,Z 188,A -132.8951,B 2.285,C 0.2398,E1 2.1794,E2 226.1084} C_DIS
LIN {X -104.9733,Y -87.4257,Z 188,A -134.762,B 2.2853,C 0.2369,E1 2.176,E2 227.9969} C_DIS
LIN {X -107.7689,Y -83.9551,Z 188,A -136.6532,B 2.2857,C 0.233,E1 2.1727,E2 229.8906} C_DIS
LIN {X -110.0399,Y -80.9551,Z 188,A -138.3742,B 2.286,C 0.23,E1 2.1698,E2 231.63} C_DIS
LIN {X -112.6602,Y -77.2669,Z 188,A -140.3566,B 2.2864,C 0.226,E1 2.1666,E2 233.623} C_DIS
LIN {X -115.1544,Y -73.4982,Z 188,A -142.3631,B 2.2868,C 0.222,E1 2.1635,E2 235.6435} C_DIS
LIN {X -117.4886,Y -69.7066,Z 188,A -144.3278,B 2.2872,C 0.2179,E1 2.1606,E2 237.6203} C_DIS
LIN {X -120.0545,Y -65.1865,Z 188,A -146.6661,B 2.2876,C 0.2131,E1 2.1574,E2 239.9785} C_DIS
LIN {X -121.7941,Y -61.872,Z 188,A -148.2009,B 2.288,C 0.2092,E1 2.1555,E2 241.508} C_DIS
LIN {X -123.3523,Y -58.7042,Z 188,A -149.782,B 2.2883,C 0.2057,E1 2.1535,E2 243.1017} C_DIS
LIN {X -124.8401,Y -55.4709,Z 188,A -151.3841,B 2.2886,C 0.2022,E1 2.1517,E2 244.7173} C_DIS
LIN {X -126.3166,Y -52.0242,Z 188,A -152.9991,B 2.289,C 0.1983,E1 2.1499,E2 246.3372} C_DIS
LIN {X -127.5055,Y -49.0362,Z 188,A -154.6208,B 2.2892,C 0.1955,E1 2.1482,E2 247.9935} C_DIS
LIN {X -128.8391,Y -45.4199,Z 188,A -156.2138,B 2.2896,C 0.1912,E1 2.1467,E2 249.5828} C_DIS
LIN {X -130.835,Y -39.3024,Z 188,A -159.0075,B 2.2901,C 0.1843,E1 2.1444,E2 252.3875} C_DIS
LIN {X -131.6704,Y -36.4016,Z 188,A -160.4702,B 2.2904,C 0.1813,E1 2.1432,E2 253.8748} C_DIS
LIN {X -132.7364,Y -32.2976,Z 188,A -162.3193,B 2.2907,C 0.1766,E1 2.142,E2 255.732} C_DIS
LIN {X -133.6007,Y -28.5127,Z 188,A -163.9718,B 2.2911,C 0.1722,E1 2.1409,E2 257.3868} C_DIS
LIN {X -134.21,Y -25.4899,Z 188,A -165.3481,B 2.2913,C 0.1689,E1 2.1402,E2 258.773} C_DIS
LIN {X -134.7616,Y -22.3912,Z 188,A -166.7693,B 2.2916,C 0.1654,E1 2.1395,E2 260.2064} C_DIS
LIN {X -135.2461,Y -19.2496,Z 188,A -168.2182,B 2.2918,C 0.162,E1 2.1389,E2 261.6693} C_DIS
LIN {X -135.7141,Y -15.6224,Z 188,A -169.8017,B 2.2921,C 0.1578,E1 2.1384,E2 263.2582} C_DIS
LIN {X -136.0127,Y -12.7556,Z 188,A -171.2501,B 2.2923,C 0.1549,E1 2.138,E2 264.7362} C_DIS
LIN {X -136.3497,Y -8.4175,Z 188,A -173.1285,B 2.2926,C 0.1499,E1 2.1376,E2 266.6203} C_DIS
LIN {X -136.5282,Y -4.7423,Z 188,A -174.8756,B 2.2929,C 0.1459,E1 2.1374,E2 268.3922} C_DIS
LIN {X -136.6119,Y -0.1256,Z 188,A -176.9552,B 2.2932,C 0.1408,E1 2.1374,E2 270.4886} C_DIS
LIN {X -136.5544,Y 3.8738,Z 188,A -178.6282,B 2.2935,C 0.1361,E1 2.1374,E2 272.1599} C_DIS
LIN {X -136.3632,Y 8.1972,Z 188,A 179.4457,B 2.2938,C 0.1312,E1 2.1377,E2 274.0988} C_DIS
LIN {X -136.102,Y 11.7642,Z 188,A 177.8625,B 2.294,C 0.1271,E1 2.1381,E2 275.6914} C_DIS
LIN {X -135.7521,Y 15.2934,Z 188,A 176.1666,B 2.2942,C 0.1234,E1 2.1386,E2 277.4124} C_DIS
LIN {X -135.2081,Y 19.5156,Z 188,A 174.4204,B 2.2945,C 0.1183,E1 2.1392,E2 279.1524} C_DIS
LIN {X -134.7183,Y 22.6508,Z 188,A 172.9353,B 2.2947,C 0.1149,E1 2.1399,E2 280.6558} C_DIS
LIN {X -133.9736,Y 26.7094,Z 188,A 171.0563,B 2.2949,C 0.1104,E1 2.1409,E2 282.5521} C_DIS
LIN {X -132.8138,Y 31.9766,Z 188,A 168.6289,B 2.2952,C 0.1046,E1 2.1424,E2 284.9984} C_DIS
LIN {X -131.9439,Y 35.3956,Z 188,A 167.1517,B 2.2953,C 0.1006,E1 2.1435,E2 286.4742} C_DIS
LIN {X -131.0634,Y 38.5281,Z 188,A 165.6107,B 2.2955,C 0.0972,E1 2.1447,E2 288.0359} C_DIS
LIN {X -129.991,Y 42.0063,Z 188,A 164.0612,B 2.2956,C 0.0932,E1 2.146,E2 289.5872} C_DIS
LIN {X -128.9712,Y 45.0389,Z 188,A 162.6532,B 2.2958,C 0.0898,E1 2.1473,E2 291.0024} C_DIS
LIN {X -127.7155,Y 48.4881,Z 188,A 160.993,B 2.2959,C 0.086,E1 2.1489,E2 292.6763} C_DIS
LIN {X -126.351,Y 51.9419,Z 188,A 159.1182,B 2.2961,C 0.0826,E1 2.1509,E2 294.5888} C_DIS
LIN {X -124.5488,Y 56.1221,Z 188,A 157.3119,B 2.2962,C 0.0776,E1 2.1529,E2 296.381} C_DIS
LIN {X -123.0855,Y 59.2627,Z 188,A 155.6497,B 2.2963,C 0.0744,E1 2.1549,E2 298.0677} C_DIS
LIN {X -121.1431,Y 63.1383,Z 188,A 153.6083,B 2.2965,C 0.0703,E1 2.1576,E2 300.1348} C_DIS
LIN {X -119.0779,Y 66.955,Z 188,A 151.8091,B 2.2965,C 0.0659,E1 2.16,E2 301.9303} C_DIS
LIN {X -116.6197,Y 71.1509,Z 188,A 149.8621,B 2.2967,C 0.0609,E1 2.1628,E2 303.8645} C_DIS
LIN {X -114.8957,Y 73.9024,Z 188,A 148.2977,B 2.2968,C 0.0582,E1 2.1651,E2 305.4525} C_DIS
LIN {X -112.5602,Y 77.4127,Z 188,A 146.4017,B 2.2968,C 0.0544,E1 2.1681,E2 307.3626} C_DIS
LIN {X -110.151,Y 80.8038,Z 188,A 144.53,B 2.297,C 0.0509,E1 2.1712,E2 309.2482} C_DIS
LIN {X -107.7767,Y 83.9451,Z 188,A 142.7806,B 2.297,C 0.0475,E1 2.1742,E2 311.0083} C_DIS
LIN {X -102.9485,Y 89.8004,Z 188,A 138.6052,B 2.2971,C 0.0434,E1 2.182,E2 315.2993} C_DIS
LIN {X -98.4881,Y 94.6717,Z 188,A 136.6928,B 2.2973,C 0.0358,E1 2.1855,E2 317.1079} C_DIS
LIN {X -92.7628,Y 100.2882,Z 188,A 133.2478,B 2.2973,C 0.0297,E1 2.1924,E2 320.5604} C_DIS
LIN {X -88.7427,Y 103.8622,Z 188,A 130.8705,B 2.2973,C 0.0261,E1 2.1974,E2 322.9507} C_DIS
LIN {X -86.0244,Y 106.1245,Z 188,A 128.7141,B 2.2973,C 0.0256,E1 2.2022,E2 325.1857} C_DIS
LIN {X -82.4787,Y 108.9022,Z 188,A 127.0546,B 2.2974,C 0.0219,E1 2.2059,E2 326.8169} C_DIS
LIN {X -78.7062,Y 111.6594,Z 188,A 125.3975,B 2.2974,C 0.018,E1 2.2095,E2 328.4367} C_DIS
LIN {X -75.8073,Y 113.6475,Z 188,A 123.7394,B 2.2974,C 0.0164,E1 2.2134,E2 330.1156} C_DIS
LIN {X -70.9028,Y 116.7705,Z 188,A 121.3623,B 2.2975,C 0.0129,E1 2.219,E2 332.484} C_DIS
LIN {X -68.0874,Y 118.4347,Z 188,A 119.3242,B 2.2975,C 0.0134,E1 2.2242,E2 334.5997} C_DIS
LIN {X -64.3232,Y 120.5204,Z 188,A 117.9693,B 2.2975,C 0.0097,E1 2.2274,E2 335.9005} C_DIS
LIN {X -61.4511,Y 122.0084,Z 188,A 116.5732,B 2.2975,C 0.0083,E1 2.2308,E2 337.3004} C_DIS
LIN {X -58.7188,Y 123.3454,Z 188,A 115.2587,B 2.2975,C 0.007,E1 2.2342,E2 338.6187} C_DIS
LIN {X -54.4048,Y 125.3081,Z 188,A 113.2024,B 2.2975,C 0.0053,E1 2.2394,E2 340.6818} C_DIS
LIN {X -51.3511,Y 126.5903,Z 188,A 111.7752,B 2.2975,C 0.0042,E1 2.2431,E2 342.1126} C_DIS
LIN {X -46.3017,Y 128.5228,Z 188,A 109.0544,B 2.2975,C 0.0041,E1 2.2504,E2 344.8852} C_DIS
LIN {X -42.2964,Y 129.8984,Z 188,A 107.7403,B 2.2975,C 0.001,E1 2.2538,E2 346.1442} C_DIS
LIN {X -39.606,Y 130.7421,Z 188,A 106.5167,B 2.2975,C 0.0003,E1 2.257,E2 347.3719} C_DIS
LIN {X -36.4063,Y 131.6691,Z 188,A 105.1206,B 2.2975,C -0.0005,E1 2.2608,E2 348.7671} C_DIS
LIN {X -33.4433,Y 132.4522,Z 188,A 103.8022,B 2.2975,C -0.0011,E1 2.2644,E2 350.0887} C_DIS
LIN {X -30.4134,Y 133.1805,Z 188,A 102.4911,B 2.2975,C -0.0017,E1 2.268,E2 351.3996} C_DIS
LIN {X -27.1929,Y 133.8752,Z 188,A 101.0754,B 2.2975,C -0.0021,E1 2.2718,E2 352.8185} C_DIS
LIN {X -23.5741,Y 134.5606,Z 188,A 99.5022,B 2.2975,C -0.0025,E1 2.2762,E2 354.3943} C_DIS
LIN {X -19.4514,Y 135.2173,Z 188,A 96.9957,B 2.2975,C 0.0005,E1 2.2834,E2 356.9881} C_DIS
LIN {X -13.6875,Y 135.9232,Z 188,A 95.3938,B 2.2975,C -0.0036,E1 2.2876,E2 358.4917} C_DIS
LIN {X -5.0429,Y 136.5165,Z 188,A 91.7746,B 2.2975,C -0.0036,E1 2.2977,E2 362.1075} C_DIS
LIN {X 1.8694,Y 136.5971,Z 188,A 88.9013,B 2.2975,C -0.0033,E1 2.3057,E2 364.9766} C_DIS
LIN {X 9.4617,Y 136.282,Z 188,A 85.7449,B 2.2975,C -0.0025,E1 2.3145,E2 368.1284} C_DIS
LIN {X 14.1514,Y 135.875,Z 188,A 83.8107,B 2.2975,C -0.0019,E1 2.3199,E2 370.0571} C_DIS
LIN {X 18.3064,Y 135.3781,Z 188,A 81.661,B 2.2975,C 0.0011,E1 2.326,E2 372.2527} C_DIS
LIN {X 23.3225,Y 134.6056,Z 188,A 79.7551,B 2.2975,C 0.0013,E1 2.3312,E2 374.1319} C_DIS
LIN {X 27.2953,Y 133.8544,Z 188,A 78.1864,B 2.2975,C 0.0017,E1 2.3354,E2 375.685} C_DIS
LIN {X 30.713,Y 133.112,Z 188,A 76.7646,B 2.2975,C 0.0026,E1 2.3393,E2 377.1011} C_DIS
LIN {X 33.6713,Y 132.3943,Z 188,A 75.4348,B 2.2975,C 0.004,E1 2.3429,E2 378.4367} C_DIS
LIN {X 37.2405,Y 131.4358,Z 188,A 73.9762,B 2.2975,C 0.0049,E1 2.3468,E2 379.8842} C_DIS
LIN {X 40.2919,Y 130.5322,Z 188,A 72.6102,B 2.2975,C 0.0064,E1 2.3505,E2 381.2536} C_DIS
LIN {X 44.9346,Y 129.0073,Z 188,A 70.6603,B 2.2975,C 0.0079,E1 2.3556,E2 383.1912} C_DIS
LIN {X 47.9114,Y 127.9315,Z 188,A 69.1879,B 2.2975,C 0.0103,E1 2.3595,E2 384.6805} C_DIS
LIN {X 51.4652,Y 126.5443,Z 188,A 67.7985,B 2.2975,C 0.0109,E1 2.3631,E2 386.0447} C_DIS
LIN {X 56.0422,Y 124.5845,Z 188,A 65.4994,B 2.2975,C 0.0149,E1 2.369,E2 388.3685} C_DIS
LIN {X 60.6593,Y 122.4028,Z 188,A 63.6846,B 2.2975,C 0.0157,E1 2.3735,E2 390.1442} C_DIS
LIN {X 63.6933,Y 120.8517,Z 188,A 62.3053,B 2.2975,C 0.0175,E1 2.3769,E2 391.5174} C_DIS
LIN {X 70.3041,Y 117.1324,Z 188,A 59.0921,B 2.2975,C 0.0225,E1 2.3847,E2 394.7343} C_DIS
LIN {X 75.0993,Y 114.1166,Z 188,A 56.8435,B 2.2974,C 0.0256,E1 2.39,E2 396.9677} C_DIS
LIN {X 78.4458,Y 111.8431,Z 188,A 55.1742,B 2.2974,C 0.0283,E1 2.3938,E2 398.6338} C_DIS
LIN {X 81.9611,Y 109.2934,Z 188,A 53.4352,B 2.2974,C 0.031,E1 2.3977,E2 400.3628} C_DIS
LIN {X 85.4412,Y 106.5948,Z 188,A 51.725,B 2.2973,C 0.0334,E1 2.4014,E2 402.0567} C_DIS
LIN {X 88.714,Y 103.8865,Z 188,A 49.9455,B 2.2973,C 0.0368,E1 2.4053,E2 403.836} C_DIS
LIN {X 94.5146,Y 98.6383,Z 188,A 46.8595,B 2.2972,C 0.042,E1 2.4116,E2 406.8989} C_DIS
LIN {X 97.778,Y 95.4049,Z 188,A 44.6455,B 2.297,C 0.048,E1 2.416,E2 409.1477} C_DIS
LIN {X 100.5417,Y 92.4871,Z 188,A 43.4176,B 2.297,C 0.0483,E1 2.4182,E2 410.3207} C_DIS
LIN {X 103.309,Y 89.3859,Z 188,A 41.7097,B 2.297,C 0.0519,E1 2.4214,E2 412.0246} C_DIS
LIN {X 106.1231,Y 86.0262,Z 188,A 39.9108,B 2.2969,C 0.0557,E1 2.4245,E2 413.8191} C_DIS
LIN {X 108.9442,Y 82.4238,Z 188,A 38.1087,B 2.2968,C 0.0592,E1 2.4276,E2 415.6073} C_DIS
LIN {X 111.6727,Y 78.6874,Z 188,A 36.2865,B 2.2967,C 0.0629,E1 2.4305,E2 417.4156} C_DIS
LIN {X 115.4228,Y 73.0761,Z 188,A 33.5855,B 2.2965,C 0.0687,E1 2.4347,E2 420.1015} C_DIS
LIN {X 118.5467,Y 67.8913,Z 188,A 31.3325,B 2.2964,C 0.0727,E1 2.4378,E2 422.3203} C_DIS
LIN {X 120.2712,Y 64.787,Z 188,A 29.7997,B 2.2963,C 0.0768,E1 2.4399,E2 423.8588} C_DIS
LIN {X 121.9587,Y 61.5486,Z 188,A 28.4008,B 2.2962,C 0.0796,E1 2.4417,E2 425.2419} C_DIS
LIN {X 123.3454,Y 58.7188,Z 188,A 27.1295,B 2.2961,C 0.0826,E1 2.4432,E2 426.5074} C_DIS
LIN {X 124.811,Y 55.5358,Z 188,A 25.7162,B 2.2959,C 0.086,E1 2.4448,E2 427.9143} C_DIS
LIN {X 126.6579,Y 51.1835,Z 188,A 23.4226,B 2.2956,C 0.0936,E1 2.4473,E2 430.2469} C_DIS
LIN {X 128.2718,Y 46.998,Z 188,A 21.9278,B 2.2956,C 0.0956,E1 2.4487,E2 431.6949} C_DIS
LIN {X 129.6821,Y 42.9485,Z 188,A 20.4249,B 2.2954,C 0.098,E1 2.45,E2 433.1618} C_DIS
LIN {X 130.733,Y 39.6359,Z 188,A 19.0702,B 2.2954,C 0.1011,E1 2.4511,E2 434.5044} C_DIS
LIN {X 131.6548,Y 36.4572,Z 188,A 17.7159,B 2.2952,C 0.1046,E1 2.4522,E2 435.8551} C_DIS
LIN {X 132.4834,Y 33.3202,Z 188,A 16.4824,B 2.295,C 0.1073,E1 2.453,E2 437.0733} C_DIS
LIN {X 133.2138,Y 30.2675,Z 188,A 15.184,B 2.2949,C 0.1108,E1 2.4538,E2 438.37} C_DIS
LIN {X 133.9972,Y 26.5935,Z 188,A 13.7328,B 2.2947,C 0.1141,E1 2.4546,E2 439.8065} C_DIS
LIN {X 134.7165,Y 22.6615,Z 188,A 12.0315,B 2.2945,C 0.119,E1 2.4555,E2 441.5118} C_DIS
LIN {X 135.4188,Y 17.9963,Z 188,A 9.6504,B 2.294,C 0.1278,E1 2.4564,E2 443.9443} C_DIS
LIN {X 136.0146,Y 12.7357,Z 188,A 7.9277,B 2.2939,C 0.1299,E1 2.4568,E2 445.606} C_DIS
LIN {X 136.4834,Y 5.8892,Z 188,A 5.5713,B 2.2936,C 0.1337,E1 2.4572,E2 447.8981} C_DIS
LIN {X 136.6006,Y -1.658,Z 188,A 2.573,B 2.2932,C 0.1413,E1 2.4573,E2 450.8772} C_DIS
LIN {X 136.4316,Y -6.9653,Z 188,A 0.4643,B 2.2929,C 0.1466,E1 2.4571,E2 452.9722} C_DIS
LIN {X 136.2339,Y -10.1211,Z 188,A -1.5051,B 2.2923,C 0.1555,E1 2.4567,E2 455.0242} C_DIS
LIN {X 135.7185,Y -15.5857,Z 188,A -2.937,B 2.2923,C 0.1548,E1 2.4563,E2 456.347} C_DIS
LIN {X 135.1799,Y -19.7128,Z 188,A -4.6592,B 2.292,C 0.1595,E1 2.4557,E2 458.0674} C_DIS
LIN {X 134.6729,Y -22.9225,Z 188,A -5.9281,B 2.2918,C 0.1625,E1 2.4551,E2 459.3252} C_DIS
LIN {X 134.0141,Y -26.5102,Z 188,A -7.4752,B 2.2915,C 0.1669,E1 2.4543,E2 460.8756} C_DIS
LIN {X 133.1871,Y -30.3844,Z 188,A -8.9726,B 2.2912,C 0.1701,E1 2.4534,E2 462.353} C_DIS
LIN {X 132.2505,Y -34.238,Z 188,A -10.5082,B 2.291,C 0.1737,E1 2.4524,E2 463.8734} C_DIS
LIN {X 131.4932,Y -37.035,Z 188,A -11.6882,B 2.2907,C 0.1767,E1 2.4515,E2 465.0496} C_DIS
LIN {X 130.2769,Y -41.1113,Z 188,A -14.2292,B 2.2899,C 0.1877,E1 2.4493,E2 467.6891} C_DIS
LIN {X 128.1098,Y -47.4354,Z 188,A -15.8919,B 2.29,C 0.1859,E1 2.4479,E2 469.207} C_DIS
LIN {X 127.0873,Y -50.112,Z 188,A -17.6881,B 2.2893,C 0.1939,E1 2.4459,E2 471.0811} C_DIS
LIN {X 125.2702,Y -54.4924,Z 188,A -19.0762,B 2.2893,C 0.1942,E1 2.4445,E2 472.3929} C_DIS
LIN {X 123.8145,Y -57.7244,Z 188,A -20.4542,B 2.2891,C 0.1972,E1 2.4429,E2 473.7579} C_DIS
LIN {X 122.1973,Y -61.0759,Z 188,A -21.9167,B 2.2888,C 0.2004,E1 2.4411,E2 475.2089} C_DIS
LIN {X 119.9466,Y -65.3859,Z 188,A -23.9281,B 2.2883,C 0.2053,E1 2.4385,E2 477.2182} C_DIS
LIN {X 117.8901,Y -69.025,Z 188,A -25.908,B 2.2878,C 0.2115,E1 2.4357,E2 479.229} C_DIS
LIN {X 115.7996,Y -72.4781,Z 188,A -27.2368,B 2.2877,C 0.2127,E1 2.4338,E2 480.5116} C_DIS
LIN {X 112.53,Y -77.4557,Z 188,A -29.5854,B 2.2872,C 0.2176,E1 2.4301,E2 482.8426} C_DIS
LIN {X 110.3738,Y -80.4996,Z 188,A -31.6094,B 2.2865,C 0.2248,E1 2.4267,E2 484.928} C_DIS
LIN {X 107.1265,Y -84.7736,Z 188,A -33.2196,B 2.2865,C 0.225,E1 2.4241,E2 486.456} C_DIS
LIN {X 104.2675,Y -88.2659,Z 188,A -34.9868,B 2.2862,C 0.2283,E1 2.421,E2 488.2082} C_DIS
LIN {X 100.1965,Y -92.861,Z 188,A -37.634,B 2.2856,C 0.2344,E1 2.416,E2 490.8669} C_DIS
LIN {X 96.8791,Y -96.3169,Z 188,A -39.3716,B 2.2853,C 0.2366,E1 2.4126,E2 492.5702} C_DIS
LIN {X 93.6474,Y -99.4619,Z 188,A -41.1627,B 2.285,C 0.2397,E1 2.4091,E2 494.3495} C_DIS
LIN {X 89.7954,Y -102.9528,Z 188,A -43.4939,B 2.2844,C 0.2451,E1 2.4041,E2 496.7024} C_DIS
LIN {X 87.1952,Y -105.1641,Z 188,A -44.4841,B 2.2844,C 0.2446,E1 2.4021,E2 497.6352} C_DIS
Enddeposition()
END
